C07302=1188.914,-2.420,-44.278,-179.914,5.732,148.990
C07303=1188.918,-2.670,-44.265,-179.916,5.731,148.990
C07304=1188.924,-2.919,-44.252,-179.918,5.732,148.991
C07305=1188.929,-3.170,-44.238,-179.921,5.731,148.992
C07306=1188.934,-3.418,-44.225,-179.923,5.731,148.992
C07307=1188.939,-3.668,-44.210,-179.926,5.730,148.993
C07308=1188.945,-3.918,-44.197,-179.928,5.729,148.993
C07309=1188.949,-4.167,-44.184,-179.931,5.729,148.994
C07310=1188.954,-4.417,-44.170,-179.934,5.728,148.995
C07311=1188.960,-4.666,-44.156,-179.936,5.727,148.995
C07312=1188.964,-4.916,-44.143,-179.938,5.727,148.996
C07313=1188.970,-5.165,-44.129,-179.941,5.726,148.997
C07314=1188.974,-5.415,-44.116,-179.944,5.726,148.997
C07315=1188.980,-5.664,-44.102,-179.946,5.725,148.998
C07316=1188.985,-5.915,-44.089,-179.948,5.725,148.999
C07317=1188.990,-6.163,-44.075,-179.951,5.725,148.999
C07318=1188.995,-6.414,-44.062,-179.953,5.725,149.000
C07319=1189.000,-6.663,-44.048,-179.955,5.724,149.000
C07320=1189.005,-6.913,-44.035,-179.958,5.723,149.001
C07321=1189.010,-7.162,-44.021,-179.961,5.723,149.002
C07322=1189.015,-7.412,-44.008,-179.963,5.722,149.002
C07323=1189.020,-7.661,-43.994,-179.966,5.721,149.003
C07324=1189.026,-7.911,-43.981,-179.968,5.721,149.004
C07325=1189.030,-8.161,-43.967,-179.971,5.720,149.004
C07326=1189.036,-8.410,-43.954,-179.974,5.720,149.005
C07327=1189.041,-8.660,-43.941,-179.975,5.720,149.005
C07328=1189.046,-8.909,-43.927,-179.978,5.719,149.006
C07329=1189.051,-9.159,-43.914,-179.980,5.719,149.007
C07330=1189.056,-9.408,-43.900,-179.983,5.719,149.008
C07331=1189.061,-9.658,-43.887,-179.986,5.718,149.008
C07332=1189.067,-9.908,-43.874,-179.988,5.717,149.009
C07333=1189.071,-10.157,-43.860,-179.991,5.717,149.009
C07334=1189.077,-10.407,-43.847,-179.993,5.716,149.010
C07335=1189.081,-10.657,-43.834,-179.996,5.716,149.011
C07336=1189.087,-10.906,-43.820,-179.997,5.716,149.011
C07337=1189.092,-11.156,-43.807,180.000,5.715,149.012
C07338=1189.097,-11.406,-43.794,179.997,5.715,149.013
C07339=1189.102,-11.654,-43.781,179.995,5.714,149.013
C07340=1189.108,-11.905,-43.767,179.992,5.714,149.014
C07341=1189.113,-12.154,-43.754,179.990,5.713,149.014
C07342=1189.118,-12.404,-43.740,179.987,5.713,149.015
C07343=1189.123,-12.653,-43.728,179.984,5.712,149.016
C07344=1189.127,-12.903,-43.715,179.983,5.712,149.016
C07345=1189.133,-13.153,-43.701,179.980,5.712,149.017
C07346=1189.137,-13.402,-43.688,179.978,5.711,149.018
C07347=1189.143,-13.652,-43.675,179.975,5.711,149.018
C07348=1189.148,-13.901,-43.662,179.973,5.710,149.019
C07349=1189.154,-14.151,-43.648,179.970,5.709,149.020
C07350=1189.158,-14.400,-43.635,179.967,5.709,149.020
C07351=1189.164,-14.650,-43.622,179.965,5.708,149.021
C07352=1189.169,-14.900,-43.609,179.963,5.708,149.021
C07353=1189.173,-15.150,-43.596,179.960,5.708,149.022
C07354=1189.179,-15.399,-43.583,179.958,5.707,149.023
C07355=1189.184,-15.648,-43.569,179.955,5.707,149.023
C07356=1189.189,-15.898,-43.556,179.953,5.707,149.024
C07357=1189.194,-16.148,-43.543,179.950,5.706,149.025
C07358=1189.199,-16.397,-43.531,179.948,5.705,149.025
C07359=1189.205,-16.647,-43.517,179.946,5.706,149.026
C07360=1189.210,-16.897,-43.504,179.943,5.705,149.027
C07361=1189.214,-17.146,-43.491,179.941,5.704,149.027
C07362=1189.220,-17.396,-43.478,179.938,5.704,149.028
C07363=1189.225,-17.645,-43.465,179.935,5.703,149.029
C07364=1189.230,-17.895,-43.452,179.933,5.703,149.029
C07365=1189.235,-18.145,-43.439,179.931,5.702,149.030
C07366=1189.241,-18.394,-43.426,179.929,5.702,149.030
C07367=1189.245,-18.644,-43.413,179.926,5.702,149.031
C07368=1189.251,-18.894,-43.400,179.923,5.701,149.032
C07369=1189.256,-19.143,-43.387,179.921,5.701,149.032
C07370=1189.260,-19.392,-43.374,179.918,5.700,149.033
C07371=1189.266,-19.642,-43.361,179.916,5.700,149.034
C07372=1189.271,-19.891,-43.348,179.914,5.700,149.034
C07373=1189.276,-20.141,-43.335,179.912,5.699,149.035
C07374=1189.282,-20.391,-43.322,179.909,5.699,149.036
C07375=1189.287,-20.640,-43.309,179.906,5.698,149.036
C07376=1189.291,-20.890,-43.296,179.904,5.698,149.037
C07377=1189.296,-21.139,-43.284,179.901,5.697,149.037
C07378=1189.302,-21.389,-43.270,179.899,5.696,149.038
C07379=1189.307,-21.639,-43.258,179.897,5.697,149.039
C07380=1189.312,-21.888,-43.245,179.894,5.696,149.039
C07381=1189.318,-22.138,-43.232,179.891,5.696,149.040
C07382=1189.322,-22.388,-43.219,179.889,5.695,149.041
C07383=1189.327,-22.637,-43.206,179.886,5.695,149.041
C07384=1189.333,-22.887,-43.194,179.884,5.694,149.042
C07385=1189.338,-23.157,-43.179,179.882,5.694,149.043
C07386=1189.343,-23.426,-43.166,179.879,5.694,149.043
C07387=1189.350,-23.696,-43.152,179.876,5.694,149.044
C07388=1189.355,-23.966,-43.138,179.874,5.693,149.045
C07389=1189.360,-24.215,-43.126,179.871,5.693,149.046
C07390=1189.365,-24.465,-43.114,179.869,5.692,149.046
C07391=1189.370,-24.715,-43.100,179.866,5.691,149.047
C07392=1189.376,-24.964,-43.087,179.864,5.691,149.047
C07393=1189.381,-25.214,-43.075,179.861,5.690,149.048
C07394=1189.386,-25.463,-43.062,179.859,5.690,149.049
C07395=1189.390,-25.713,-43.049,179.857,5.690,149.049
C07396=1189.396,-25.963,-43.036,179.854,5.689,149.050
C07397=1189.401,-26.212,-43.023,179.851,5.689,149.051
C07398=1189.407,-26.462,-43.012,179.849,5.688,149.051
C07399=1189.411,-26.712,-42.999,179.847,5.689,149.052
C07400=1189.416,-26.961,-42.986,179.844,5.688,149.052
C07401=1189.422,-27.211,-42.973,179.842,5.688,149.053
C07402=1189.427,-27.460,-42.961,179.840,5.687,149.054
C07403=1189.431,-27.710,-42.948,179.837,5.686,149.054
C07404=1189.437,-27.960,-42.935,179.835,5.687,149.055
C07405=1189.442,-28.210,-42.923,179.832,5.686,149.056
C07406=1189.448,-28.459,-42.910,179.830,5.685,149.056
C07407=1189.453,-28.708,-42.897,179.827,5.685,149.057
C07408=1189.457,-28.958,-42.885,179.825,5.684,149.058
C07409=1189.463,-29.208,-42.873,179.823,5.685,149.058
C07410=1189.468,-29.457,-42.860,179.820,5.684,149.059
C07411=1189.473,-29.707,-42.847,179.818,5.684,149.059
C07412=1189.478,-29.956,-42.835,179.815,5.683,149.060
C07413=1189.483,-30.207,-42.823,179.812,5.683,149.061
C07414=1189.489,-30.456,-42.809,179.810,5.683,149.062
C07415=1189.494,-30.706,-42.797,179.808,5.682,149.062
C07416=1189.499,-30.956,-42.785,179.806,5.682,149.063
C07417=1189.504,-31.205,-42.772,179.803,5.681,149.063
C07418=1189.509,-31.455,-42.759,179.800,5.681,149.064
C07419=1189.514,-31.704,-42.747,179.799,5.681,149.065
C07420=1189.519,-31.954,-42.735,179.796,5.680,149.065
C07421=1189.525,-32.204,-42.722,179.793,5.680,149.066
C07422=1189.530,-32.453,-42.710,179.791,5.679,149.067
C07423=1189.535,-32.703,-42.698,179.788,5.679,149.067
C07424=1189.540,-32.952,-42.685,179.786,5.679,149.068
C07425=1189.545,-33.202,-42.672,179.784,5.678,149.069
C07426=1189.550,-33.452,-42.660,179.781,5.678,149.069
C07427=1189.555,-33.701,-42.648,179.779,5.677,149.070
C07428=1189.561,-33.951,-42.636,179.776,5.677,149.070
C07429=1189.566,-34.201,-42.623,179.774,5.677,149.071
C07430=1189.571,-34.450,-42.611,179.772,5.677,149.072
C07431=1189.576,-34.700,-42.599,179.769,5.676,149.073
C07432=1189.582,-34.949,-42.586,179.767,5.675,149.073
C07433=1189.586,-35.200,-42.574,179.765,5.676,149.074
C07434=1189.592,-35.449,-42.561,179.762,5.675,149.074
C07435=1189.597,-35.698,-42.549,179.759,5.675,149.075
C07436=1189.602,-35.948,-42.537,179.757,5.674,149.076
C07437=1189.607,-36.198,-42.524,179.755,5.674,149.076
C07438=1189.613,-36.448,-42.512,179.752,5.674,149.077
C07439=1189.617,-36.697,-42.500,179.750,5.673,149.078
C07440=1189.622,-36.947,-42.488,179.748,5.673,149.078
C07441=1189.628,-37.196,-42.476,179.745,5.672,149.079
C07442=1189.633,-37.446,-42.464,179.743,5.672,149.080
C07443=1189.638,-37.695,-42.451,179.740,5.672,149.080
C07444=1189.644,-37.945,-42.439,179.738,5.671,149.081
C07445=1189.648,-38.195,-42.426,179.735,5.671,149.081
C07446=1189.654,-38.445,-42.415,179.733,5.671,149.082
C07447=1189.659,-38.694,-42.402,179.731,5.671,149.083
C07448=1189.664,-38.944,-42.390,179.728,5.670,149.083
C07449=1189.669,-39.194,-42.378,179.726,5.669,149.084
C07450=1189.674,-39.443,-42.366,179.724,5.670,149.085
C07451=1189.679,-39.693,-42.354,179.721,5.669,149.085
C07452=1189.684,-39.943,-42.342,179.719,5.668,149.086
C07453=1189.690,-40.192,-42.330,179.716,5.668,149.087
C07454=1189.695,-40.442,-42.317,179.714,5.668,149.087
C07455=1189.700,-40.692,-42.305,179.711,5.668,149.088
C07456=1189.706,-40.941,-42.293,179.709,5.667,149.088
C07457=1189.710,-41.191,-42.281,179.707,5.667,149.089
C07458=1189.716,-41.441,-42.270,179.704,5.667,149.090
C07459=1189.721,-41.690,-42.257,179.702,5.667,149.091
C07460=1189.726,-41.940,-42.245,179.700,5.666,149.091
C07461=1189.731,-42.189,-42.233,179.697,5.665,149.092
C07462=1189.736,-42.439,-42.221,179.695,5.666,149.092
C07463=1189.741,-42.689,-42.209,179.692,5.665,149.093
C07464=1189.747,-42.938,-42.197,179.690,5.665,149.094
C07465=1189.752,-43.188,-42.185,179.687,5.664,149.094
C07466=1189.757,-43.438,-42.173,179.685,5.664,149.095
C07467=1189.762,-43.687,-42.161,179.683,5.664,149.096
C07468=1189.767,-43.937,-42.149,179.680,5.663,149.096
C07469=1189.773,-44.187,-42.137,179.678,5.663,149.097
C07470=1189.778,-44.436,-42.125,179.676,5.663,149.098
C07471=1189.783,-44.686,-42.113,179.673,5.663,149.098
C07472=1189.788,-44.936,-42.101,179.670,5.662,149.099
C07473=1189.793,-45.186,-42.090,179.668,5.661,149.099
C07474=1189.799,-45.435,-42.077,179.666,5.662,149.100
C07475=1189.803,-45.685,-42.066,179.663,5.661,149.101
C07476=1189.809,-45.934,-42.054,179.661,5.661,149.102
C07477=1189.814,-46.184,-42.041,179.659,5.661,149.102
C07478=1189.819,-46.434,-42.029,179.657,5.660,149.103
C07479=1189.824,-46.683,-42.018,179.654,5.660,149.103
C07480=1189.829,-46.933,-42.006,179.651,5.659,149.104
C07481=1189.835,-47.183,-41.994,179.650,5.659,149.105
C07482=1189.839,-47.432,-41.982,179.647,5.659,149.105
C07483=1189.845,-47.681,-41.971,179.644,5.658,149.106
C07484=1189.851,-47.931,-41.959,179.642,5.658,149.107
C07485=1189.856,-48.181,-41.947,179.640,5.658,149.107
C07486=1189.861,-48.431,-41.936,179.637,5.658,149.108
C07487=1189.866,-48.680,-41.923,179.635,5.657,149.109
C07488=1189.871,-48.930,-41.911,179.633,5.657,149.109
C07489=1189.877,-49.201,-41.898,179.630,5.657,149.110
C07490=1189.883,-49.471,-41.886,179.628,5.656,149.110
C07491=1189.888,-49.741,-41.873,179.625,5.656,149.111
C07492=1189.893,-50.012,-41.860,179.622,5.655,149.112
C07493=1189.899,-50.260,-41.849,179.620,5.655,149.113
C07494=1189.904,-50.510,-41.838,179.618,5.655,149.113
C07495=1189.910,-50.760,-41.826,179.615,5.655,149.114
C07496=1189.914,-51.009,-41.814,179.613,5.654,149.114
C07497=1189.919,-51.259,-41.802,179.611,5.654,149.115
C07498=1189.925,-51.509,-41.790,179.608,5.654,149.116
C07499=1189.929,-51.759,-41.779,179.605,5.654,149.117
C07500=1189.935,-52.009,-41.767,179.603,5.653,149.117
C07501=1189.940,-52.258,-41.756,179.601,5.653,149.118
C07502=1189.946,-52.508,-41.744,179.598,5.653,149.118
C07503=1189.950,-52.757,-41.733,179.596,5.652,149.119
C07504=1189.956,-53.007,-41.721,179.594,5.652,149.120
C07505=1189.961,-53.257,-41.709,179.592,5.652,149.120
C07506=1189.966,-53.507,-41.698,179.589,5.651,149.121
C07507=1189.971,-53.757,-41.686,179.587,5.652,149.122
C07508=1189.977,-54.006,-41.675,179.585,5.651,149.122
C07509=1189.982,-54.256,-41.663,179.582,5.650,149.123
C07510=1189.987,-54.505,-41.652,179.579,5.650,149.124
C07511=1189.992,-54.755,-41.640,179.577,5.650,149.124
C07512=1189.997,-55.005,-41.628,179.575,5.650,149.125
C07513=1190.002,-55.255,-41.616,179.572,5.649,149.125
C07514=1190.008,-55.505,-41.605,179.570,5.649,149.126
C07515=1190.013,-55.754,-41.594,179.568,5.649,149.127
C07516=1190.018,-56.004,-41.582,179.565,5.648,149.127
C07517=1190.023,-56.253,-41.571,179.563,5.649,149.128
C07518=1190.029,-56.503,-41.559,179.561,5.648,149.129
C07519=1190.033,-56.753,-41.547,179.558,5.647,149.129
C07520=1190.039,-57.002,-41.536,179.556,5.648,149.130
C07521=1190.044,-57.252,-41.525,179.554,5.647,149.131
C07522=1190.049,-57.501,-41.513,179.551,5.647,149.131
C07523=1190.054,-57.751,-41.501,179.549,5.646,149.132
C07524=1190.059,-58.001,-41.490,179.547,5.646,149.133
C07525=1190.065,-58.250,-41.479,179.544,5.646,149.133
C07526=1190.070,-58.500,-41.468,179.541,5.645,149.134
C07527=1190.075,-58.750,-41.456,179.540,5.645,149.134
C07528=1190.080,-59.000,-41.445,179.537,5.645,149.135
C07529=1190.085,-59.250,-41.433,179.535,5.645,149.136
C07530=1190.091,-59.499,-41.422,179.532,5.645,149.137
C07531=1190.096,-59.749,-41.410,179.530,5.644,149.137
C07532=1190.101,-59.998,-41.399,179.528,5.644,149.138
C07533=1190.105,-60.248,-41.388,179.526,5.644,149.138
C07534=1190.112,-60.498,-41.377,179.523,5.643,149.139
C07535=1190.116,-60.747,-41.365,179.521,5.643,149.140
C07536=1190.122,-60.997,-41.354,179.519,5.643,149.140
C07537=1190.127,-61.247,-41.342,179.516,5.643,149.141
C07538=1190.132,-61.496,-41.331,179.514,5.642,149.142
C07539=1190.138,-61.746,-41.320,179.512,5.642,149.142
C07540=1190.142,-61.996,-41.309,179.509,5.642,149.143
C07541=1190.148,-62.246,-41.297,179.506,5.641,149.144
C07542=1190.153,-62.495,-41.286,179.505,5.641,149.144
C07543=1190.158,-62.744,-41.275,179.502,5.641,149.145
C07544=1190.163,-62.995,-41.264,179.499,5.641,149.146
C07545=1190.169,-63.244,-41.253,179.498,5.641,149.146
C07546=1190.174,-63.494,-41.241,179.495,5.640,149.147
C07547=1190.179,-63.744,-41.229,179.492,5.640,149.147
C07548=1190.184,-63.994,-41.219,179.490,5.640,149.148
C07549=1190.190,-64.243,-41.207,179.488,5.639,149.149
C07550=1190.195,-64.493,-41.196,179.486,5.639,149.149
C07551=1190.200,-64.743,-41.186,179.483,5.639,149.150
C07552=1190.206,-64.992,-41.174,179.481,5.639,149.151
C07553=1190.210,-65.242,-41.163,179.479,5.638,149.151
C07554=1190.215,-65.492,-41.152,179.477,5.638,149.152
C07555=1190.221,-65.741,-41.141,179.474,5.638,149.153
C07556=1190.226,-65.991,-41.129,179.472,5.637,149.153
C07557=1190.231,-66.241,-41.119,179.470,5.638,149.154
C07558=1190.236,-66.490,-41.108,179.467,5.637,149.154
C07559=1190.242,-66.740,-41.096,179.464,5.637,149.155
C07560=1190.247,-66.990,-41.085,179.463,5.637,149.156
C07561=1190.252,-67.239,-41.074,179.460,5.636,149.156
C07562=1190.257,-67.489,-41.063,179.457,5.636,149.157
C07563=1190.262,-67.739,-41.052,179.456,5.636,149.158
C07564=1190.268,-67.988,-41.041,179.453,5.635,149.158
C07565=1190.272,-68.238,-41.030,179.451,5.636,149.159
C07566=1190.278,-68.488,-41.019,179.448,5.635,149.160
C07567=1190.284,-68.737,-41.008,179.446,5.635,149.160
C07568=1190.289,-68.988,-40.997,179.444,5.635,149.161
C07569=1190.295,-69.237,-40.986,179.441,5.634,149.162
C07570=1190.299,-69.486,-40.974,179.439,5.634,149.162
C07571=1190.304,-69.737,-40.964,179.437,5.634,149.163
C07572=1190.310,-69.986,-40.953,179.434,5.634,149.163
C07573=1190.315,-70.236,-40.942,179.432,5.633,149.164
C07574=1190.320,-70.486,-40.930,179.430,5.633,149.165
C07575=1190.326,-70.735,-40.920,179.427,5.633,149.165
C07576=1190.330,-70.985,-40.909,179.425,5.633,149.166
C07577=1190.336,-71.234,-40.899,179.423,5.632,149.167
C07578=1190.341,-71.484,-40.887,179.421,5.632,149.167
C07579=1190.346,-71.735,-40.876,179.418,5.632,149.168
C07580=1190.352,-71.984,-40.865,179.416,5.632,149.169
C07581=1190.357,-72.234,-40.855,179.414,5.631,149.169
C07582=1190.362,-72.483,-40.844,179.412,5.631,149.170
C07583=1190.368,-72.733,-40.833,179.409,5.631,149.171
C07584=1190.373,-72.982,-40.822,179.407,5.630,149.171
C07585=1190.378,-73.232,-40.811,179.405,5.631,149.172
C07586=1190.383,-73.482,-40.800,179.402,5.630,149.172
C07587=1190.388,-73.732,-40.790,179.400,5.631,149.173
C07588=1190.393,-73.981,-40.778,179.398,5.630,149.174
C07589=1190.398,-74.231,-40.768,179.395,5.629,149.174
C07590=1190.404,-74.481,-40.757,179.393,5.630,149.175
C07591=1190.409,-74.730,-40.746,179.391,5.629,149.176
C07592=1190.414,-74.981,-40.735,179.388,5.628,149.176
C07593=1190.420,-75.252,-40.723,179.386,5.629,149.177
C07594=1190.426,-75.521,-40.712,179.383,5.628,149.178
C07595=1190.431,-75.793,-40.700,179.381,5.628,149.178
C07596=1190.437,-76.064,-40.688,179.378,5.628,149.179
C07597=1190.443,-76.314,-40.678,179.376,5.628,149.180
C07598=1190.447,-76.563,-40.667,179.374,5.627,149.180
C07599=1190.453,-76.813,-40.656,179.372,5.628,149.181
C07600=1190.458,-77.063,-40.646,179.369,5.627,149.182
C07601=1190.463,-77.312,-40.635,179.367,5.626,149.182
C07602=1190.468,-77.562,-40.624,179.365,5.627,149.183
C07603=1190.474,-77.812,-40.614,179.362,5.626,149.184
C07604=1190.479,-78.061,-40.603,179.360,5.626,149.184
C07605=1190.484,-78.311,-40.593,179.358,5.626,149.185
C07606=1190.490,-78.561,-40.581,179.355,5.625,149.186
C07607=1190.495,-78.810,-40.571,179.353,5.625,149.186
C07608=1190.500,-79.061,-40.560,179.351,5.625,149.187
C07609=1190.506,-79.310,-40.550,179.348,5.625,149.187
C07610=1190.510,-79.560,-40.538,179.347,5.625,149.188
C07611=1190.516,-79.809,-40.528,179.344,5.624,149.189
C07612=1190.521,-80.060,-40.518,179.342,5.625,149.189
C07613=1190.527,-80.309,-40.507,179.339,5.624,149.190
C07614=1190.531,-80.559,-40.496,179.337,5.623,149.190
C07615=1190.537,-80.808,-40.486,179.335,5.624,149.191
C07616=1190.542,-81.059,-40.475,179.332,5.623,149.192
C07617=1190.548,-81.308,-40.465,179.331,5.623,149.192
C07618=1190.553,-81.557,-40.454,179.328,5.623,149.193
C07619=1190.558,-81.807,-40.444,179.325,5.622,149.194
C07620=1190.563,-82.057,-40.433,179.324,5.622,149.194
C07621=1190.568,-82.307,-40.423,179.321,5.622,149.195
C07622=1190.574,-82.557,-40.413,179.319,5.622,149.196
C07623=1190.579,-82.806,-40.401,179.317,5.622,149.196
C07624=1190.584,-83.056,-40.391,179.315,5.622,149.197
C07625=1190.589,-83.306,-40.381,179.312,5.622,149.198
C07626=1190.595,-83.556,-40.370,179.310,5.621,149.198
C07627=1190.601,-83.805,-40.360,179.308,5.621,149.199
C07628=1190.604,-84.054,-40.349,179.305,5.621,149.200
C07629=1190.610,-84.304,-40.339,179.303,5.621,149.200
C07630=1190.615,-84.554,-40.329,179.301,5.620,149.201
C07631=1190.621,-84.804,-40.319,179.298,5.620,149.201
C07632=1190.626,-85.054,-40.308,179.296,5.620,149.202
C07633=1190.631,-85.304,-40.298,179.294,5.620,149.203
C07634=1190.637,-85.553,-40.288,179.292,5.620,149.203
C07635=1190.642,-85.803,-40.276,179.289,5.619,149.204
C07636=1190.647,-86.052,-40.266,179.287,5.619,149.205
C07637=1190.652,-86.302,-40.255,179.285,5.619,149.205
C07638=1190.658,-86.552,-40.245,179.283,5.618,149.206
C07639=1190.663,-86.801,-40.236,179.280,5.619,149.206
C07640=1190.668,-87.052,-40.225,179.278,5.618,149.207
C07641=1190.673,-87.301,-40.215,179.276,5.618,149.208
C07642=1190.678,-87.551,-40.204,179.274,5.618,149.208
C07643=1190.684,-87.801,-40.194,179.271,5.617,149.209
C07644=1190.689,-88.050,-40.184,179.269,5.617,149.209
C07645=1190.694,-88.301,-40.173,179.267,5.617,149.210
C07646=1190.700,-88.550,-40.163,179.264,5.617,149.211
C07647=1190.705,-88.799,-40.153,179.262,5.617,149.211
C07648=1190.710,-89.050,-40.143,179.260,5.616,149.212
C07649=1190.715,-89.299,-40.133,179.258,5.617,149.213
C07650=1190.720,-89.549,-40.122,179.255,5.616,149.213
C07651=1190.726,-89.798,-40.111,179.253,5.616,149.214
C07652=1190.731,-90.048,-40.101,179.251,5.616,149.215
C07653=1190.736,-90.298,-40.092,179.249,5.616,149.215
C07654=1190.742,-90.548,-40.081,179.246,5.615,149.216
C07655=1190.747,-90.798,-40.071,179.244,5.615,149.217
C07656=1190.752,-91.048,-40.061,179.242,5.615,149.217
C07657=1190.758,-91.297,-40.050,179.239,5.615,149.218
C07658=1190.763,-91.547,-40.041,179.237,5.615,149.219
C07659=1190.768,-91.797,-40.030,179.235,5.614,149.219
C07660=1190.773,-92.046,-40.020,179.233,5.615,149.220
C07661=1190.779,-92.296,-40.010,179.230,5.614,149.220
C07662=1190.784,-92.546,-39.999,179.229,5.614,149.221
C07663=1190.789,-92.795,-39.990,179.226,5.614,149.222
C07664=1190.794,-93.045,-39.979,179.223,5.613,149.222
C07665=1190.799,-93.295,-39.969,179.222,5.613,149.223
C07666=1190.805,-93.545,-39.959,179.219,5.613,149.224
C07667=1190.810,-93.794,-39.949,179.217,5.613,149.224
C07668=1190.815,-94.043,-39.939,179.215,5.613,149.225
C07669=1190.821,-94.294,-39.929,179.213,5.613,149.225
C07670=1190.826,-94.544,-39.919,179.210,5.613,149.226
C07671=1190.831,-94.793,-39.909,179.209,5.613,149.227
C07672=1190.836,-95.043,-39.899,179.206,5.612,149.227
C07673=1190.842,-95.293,-39.888,179.204,5.611,149.228
C07674=1190.847,-95.542,-39.878,179.202,5.612,149.229
C07675=1190.852,-95.792,-39.869,179.199,5.611,149.229
C07676=1190.857,-96.043,-39.859,179.197,5.611,149.230
C07677=1190.863,-96.292,-39.849,179.195,5.611,149.230
C07678=1190.868,-96.541,-39.839,179.193,5.611,149.231
C07679=1190.873,-96.791,-39.829,179.190,5.611,149.232
C07680=1190.878,-97.041,-39.818,179.188,5.611,149.232
C07681=1190.884,-97.291,-39.808,179.186,5.611,149.233
C07682=1190.889,-97.540,-39.799,179.183,5.610,149.234
C07683=1190.895,-97.790,-39.789,179.181,5.610,149.234
C07684=1190.900,-98.040,-39.778,179.179,5.609,149.235
C07685=1190.905,-98.290,-39.769,179.177,5.610,149.235
C07686=1190.911,-98.540,-39.759,179.174,5.609,149.236
C07687=1190.916,-98.789,-39.749,179.173,5.609,149.237
C07688=1190.920,-99.039,-39.739,179.170,5.609,149.237
C07689=1190.926,-99.289,-39.729,179.168,5.609,149.238
C07690=1190.932,-99.539,-39.719,179.166,5.609,149.239
C07691=1190.937,-99.788,-39.710,179.164,5.609,149.239
C07692=1190.942,-100.038,-39.699,179.162,5.608,149.240
C07693=1190.947,-100.288,-39.689,179.159,5.608,149.240
C07694=1190.953,-100.538,-39.680,179.157,5.608,149.241
C07695=1190.958,-100.787,-39.670,179.155,5.607,149.242
C07696=1190.963,-101.037,-39.660,179.153,5.608,149.242
C07697=1190.969,-101.309,-39.649,179.150,5.607,149.243
C07698=1190.974,-101.580,-39.638,179.148,5.608,149.244
C07699=1190.980,-101.852,-39.628,179.146,5.607,149.244
C07700=1190.986,-102.123,-39.617,179.143,5.607,149.245
C07701=1190.991,-102.373,-39.608,179.141,5.607,149.246
C07702=1190.997,-102.623,-39.597,179.138,5.607,149.246
C07703=1191.001,-102.872,-39.588,179.137,5.607,149.247
C07704=1191.007,-103.122,-39.578,179.134,5.606,149.248
C07705=1191.012,-103.372,-39.569,179.132,5.606,149.248
C07706=1191.018,-103.621,-39.559,179.130,5.606,149.249
C07707=1191.022,-103.872,-39.549,179.127,5.605,149.250
C07708=1191.028,-104.121,-39.539,179.125,5.605,149.250
C07709=1191.034,-104.371,-39.530,179.123,5.605,149.251
C07710=1191.039,-104.621,-39.520,179.121,5.605,149.251
C07711=1191.044,-104.870,-39.510,179.118,5.605,149.252
C07712=1191.050,-105.120,-39.501,179.116,5.605,149.253
C07713=1191.055,-105.370,-39.490,179.114,5.604,149.253
C07714=1191.060,-105.620,-39.481,179.112,5.605,149.254
C07715=1191.065,-105.870,-39.471,179.110,5.604,149.254
C07716=1191.070,-106.119,-39.462,179.108,5.604,149.255
C07717=1191.076,-106.369,-39.452,179.105,5.604,149.256
C07718=1191.081,-106.618,-39.442,179.103,5.604,149.256
C07719=1191.087,-106.868,-39.433,179.101,5.603,149.257
C07720=1191.091,-107.118,-39.423,179.099,5.603,149.257
C07721=1191.097,-107.369,-39.414,179.096,5.603,149.258
C07722=1191.102,-107.618,-39.404,179.094,5.603,149.259
C07723=1191.108,-107.868,-39.394,179.092,5.603,149.259
C07724=1191.113,-108.117,-39.385,179.090,5.603,149.260
C07725=1191.119,-108.367,-39.375,179.088,5.602,149.261
C07726=1191.123,-108.617,-39.366,179.086,5.603,149.261
C07727=1191.129,-108.867,-39.356,179.083,5.602,149.262
C07728=1191.134,-109.116,-39.347,179.081,5.601,149.262
C07729=1191.139,-109.366,-39.338,179.079,5.602,149.263
C07730=1191.144,-109.616,-39.327,179.077,5.601,149.264
C07731=1191.149,-109.866,-39.318,179.075,5.601,149.264
C07732=1191.155,-110.115,-39.308,179.072,5.601,149.265
C07733=1191.160,-110.365,-39.299,179.070,5.601,149.266
C07734=1191.166,-110.615,-39.289,179.068,5.601,149.266
C07735=1191.171,-110.865,-39.280,179.066,5.601,149.267
C07736=1191.177,-111.114,-39.270,179.063,5.600,149.268
C07737=1191.182,-111.364,-39.261,179.062,5.600,149.268
C07738=1191.187,-111.614,-39.252,179.059,5.600,149.269
C07739=1191.193,-111.863,-39.242,179.057,5.600,149.269
C07740=1191.198,-112.113,-39.233,179.055,5.600,149.270
C07741=1191.203,-112.363,-39.223,179.053,5.600,149.271
C07742=1191.208,-112.613,-39.214,179.051,5.599,149.271
C07743=1191.214,-112.863,-39.205,179.048,5.600,149.272
C07744=1191.219,-113.113,-39.194,179.046,5.599,149.273
C07745=1191.224,-113.363,-39.185,179.044,5.599,149.273
C07746=1191.229,-113.612,-39.176,179.041,5.599,149.274
C07747=1191.235,-113.862,-39.166,179.040,5.599,149.274
C07748=1191.240,-114.112,-39.157,179.037,5.598,149.275
C07749=1191.245,-114.361,-39.147,179.036,5.598,149.275
C07750=1191.250,-114.611,-39.138,179.033,5.598,149.276
C07751=1191.256,-114.861,-39.129,179.031,5.598,149.277
C07752=1191.261,-115.111,-39.119,179.029,5.598,149.277
C07753=1191.266,-115.361,-39.110,179.027,5.598,149.278
C07754=1191.272,-115.610,-39.101,179.024,5.597,149.279
C07755=1191.277,-115.860,-39.091,179.022,5.598,149.279
C07756=1191.282,-116.110,-39.082,179.020,5.597,149.280
C07757=1191.288,-116.360,-39.073,179.018,5.597,149.280
C07758=1191.293,-116.610,-39.064,179.016,5.597,149.281
C07759=1191.298,-116.859,-39.054,179.014,5.597,149.282
C07760=1191.303,-117.109,-39.045,179.011,5.597,149.282
C07761=1191.309,-117.359,-39.036,179.009,5.597,149.283
C07762=1191.314,-117.608,-39.026,179.007,5.596,149.284
C07763=1191.319,-117.858,-39.017,179.005,5.596,149.284
C07764=1191.325,-118.108,-39.008,179.003,5.596,149.285
C07765=1191.330,-118.358,-38.999,179.001,5.596,149.285
C07766=1191.335,-118.607,-38.989,178.998,5.595,149.286
C07767=1191.340,-118.857,-38.980,178.997,5.595,149.286
C07768=1191.346,-119.107,-38.971,178.994,5.595,149.287
C07769=1191.352,-119.357,-38.962,178.992,5.595,149.288
C07770=1191.357,-119.607,-38.953,178.990,5.595,149.288
C07771=1191.362,-119.856,-38.944,178.988,5.595,149.289
C07772=1191.367,-120.107,-38.934,178.986,5.595,149.290
C07773=1191.373,-120.356,-38.926,178.983,5.595,149.290
C07774=1191.378,-120.606,-38.917,178.982,5.595,149.291
C07775=1191.384,-120.855,-38.908,178.979,5.594,149.292
C07776=1191.388,-121.105,-38.898,178.977,5.594,149.292
C07777=1191.394,-121.355,-38.889,178.975,5.594,149.293
C07778=1191.400,-121.605,-38.880,178.973,5.594,149.293
C07779=1191.405,-121.854,-38.871,178.970,5.594,149.294
C07780=1191.410,-122.104,-38.862,178.969,5.594,149.294
C07781=1191.416,-122.354,-38.852,178.966,5.593,149.295
C07782=1191.421,-122.604,-38.843,178.965,5.593,149.296
C07783=1191.426,-122.854,-38.834,178.962,5.593,149.296
C07784=1191.431,-123.103,-38.825,178.960,5.593,149.297
C07785=1191.436,-123.353,-38.816,178.958,5.592,149.298
C07786=1191.442,-123.603,-38.807,178.956,5.593,149.298
C07787=1191.447,-123.853,-38.798,178.953,5.592,149.299
C07788=1191.453,-124.102,-38.789,178.951,5.593,149.299
C07789=1191.458,-124.352,-38.780,178.949,5.592,149.300
C07790=1191.463,-124.602,-38.771,178.947,5.592,149.301
C07791=1191.468,-124.851,-38.762,178.945,5.591,149.301
C07792=1191.474,-125.102,-38.752,178.943,5.592,149.302
C07793=1191.479,-125.351,-38.743,178.941,5.591,149.302
C07794=1191.484,-125.601,-38.735,178.938,5.591,149.303
C07795=1191.490,-125.851,-38.726,178.937,5.591,149.304
C07796=1191.495,-126.101,-38.717,178.934,5.591,149.304
C07797=1191.500,-126.350,-38.708,178.933,5.591,149.305
C07798=1191.506,-126.600,-38.699,178.930,5.591,149.305
C07799=1191.512,-126.850,-38.690,178.928,5.591,149.306
C07800=1191.517,-127.100,-38.681,178.926,5.590,149.307
C07801=1191.095,-127.111,-38.720,178.922,5.594,149.309
C07802=1191.090,-126.861,-38.729,178.924,5.594,149.308
C07803=1191.084,-126.611,-38.738,178.926,5.594,149.307
C07804=1191.079,-126.361,-38.747,178.929,5.594,149.307
C07805=1191.074,-126.111,-38.756,178.930,5.594,149.306
C07806=1191.068,-125.862,-38.764,178.933,5.595,149.305
C07807=1191.063,-125.612,-38.773,178.935,5.595,149.305
C07808=1191.058,-125.363,-38.783,178.937,5.595,149.304
C07809=1191.052,-125.113,-38.792,178.939,5.595,149.304
C07810=1191.047,-124.863,-38.801,178.941,5.595,149.303
C07811=1191.042,-124.613,-38.810,178.943,5.595,149.302
C07812=1191.037,-124.363,-38.819,178.946,5.596,149.302
C07813=1191.032,-124.113,-38.828,178.947,5.596,149.301
C07814=1191.026,-123.863,-38.837,178.949,5.595,149.301
C07815=1191.021,-123.613,-38.846,178.952,5.596,149.300
C07816=1191.015,-123.364,-38.855,178.954,5.596,149.299
C07817=1191.010,-123.114,-38.864,178.956,5.596,149.299
C07818=1191.004,-122.865,-38.873,178.958,5.596,149.298
C07819=1191.000,-122.615,-38.882,178.960,5.597,149.298
C07820=1190.994,-122.365,-38.892,178.962,5.596,149.297
C07821=1190.989,-122.115,-38.901,178.964,5.597,149.296
C07822=1190.983,-121.865,-38.910,178.967,5.597,149.296
C07823=1190.978,-121.616,-38.919,178.969,5.598,149.295
C07824=1190.972,-121.365,-38.928,178.971,5.597,149.295
C07825=1190.967,-121.116,-38.937,178.973,5.598,149.294
C07826=1190.962,-120.866,-38.947,178.975,5.598,149.293
C07827=1190.957,-120.616,-38.955,178.978,5.598,149.293
C07828=1190.952,-120.367,-38.964,178.979,5.598,149.292
C07829=1190.946,-120.116,-38.974,178.982,5.598,149.291
C07830=1190.941,-119.867,-38.983,178.984,5.598,149.291
C07831=1190.935,-119.618,-38.992,178.986,5.599,149.290
C07832=1190.930,-119.368,-39.001,178.988,5.599,149.290
C07833=1190.924,-119.118,-39.010,178.991,5.599,149.289
C07834=1190.919,-118.868,-39.019,178.992,5.599,149.289
C07835=1190.914,-118.618,-39.028,178.995,5.599,149.288
C07836=1190.909,-118.369,-39.038,178.997,5.599,149.287
C07837=1190.903,-118.119,-39.047,178.999,5.600,149.287
C07838=1190.898,-117.869,-39.056,179.001,5.599,149.286
C07839=1190.893,-117.619,-39.065,179.003,5.600,149.285
C07840=1190.887,-117.370,-39.075,179.006,5.600,149.285
C07841=1190.882,-117.120,-39.084,179.008,5.601,149.284
C07842=1190.877,-116.870,-39.093,179.010,5.600,149.284
C07843=1190.872,-116.621,-39.103,179.012,5.601,149.283
C07844=1190.866,-116.371,-39.112,179.014,5.600,149.282
C07845=1190.861,-116.121,-39.121,179.016,5.601,149.282
C07846=1190.856,-115.871,-39.130,179.018,5.601,149.281
C07847=1190.850,-115.621,-39.140,179.021,5.602,149.281
C07848=1190.845,-115.372,-39.149,179.023,5.601,149.280
C07849=1190.840,-115.122,-39.158,179.025,5.601,149.279
C07850=1190.834,-114.872,-39.168,179.027,5.602,149.279
C07851=1190.829,-114.622,-39.177,179.029,5.601,149.278
C07852=1190.823,-114.372,-39.187,179.031,5.602,149.278
C07853=1190.818,-114.123,-39.196,179.033,5.602,149.277
C07854=1190.813,-113.873,-39.205,179.035,5.602,149.276
C07855=1190.807,-113.623,-39.215,179.038,5.602,149.276
C07856=1190.803,-113.374,-39.224,179.040,5.602,149.275
C07857=1190.797,-113.124,-39.233,179.042,5.603,149.274
C07858=1190.792,-112.873,-39.243,179.045,5.603,149.274
C07859=1190.787,-112.624,-39.253,179.047,5.604,149.273
C07860=1190.781,-112.374,-39.262,179.049,5.603,149.272
C07861=1190.776,-112.124,-39.272,179.051,5.604,149.272
C07862=1190.771,-111.874,-39.281,179.053,5.604,149.271
C07863=1190.765,-111.624,-39.290,179.056,5.604,149.271
C07864=1190.760,-111.375,-39.300,179.057,5.604,149.270
C07865=1190.755,-111.125,-39.309,179.060,5.604,149.269
C07866=1190.750,-110.876,-39.319,179.062,5.604,149.269
C07867=1190.745,-110.626,-39.328,179.064,5.605,149.268
C07868=1190.739,-110.376,-39.338,179.066,5.605,149.268
C07869=1190.734,-110.126,-39.347,179.069,5.605,149.267
C07870=1190.728,-109.877,-39.357,179.071,5.605,149.266
C07871=1190.723,-109.627,-39.366,179.073,5.605,149.266
C07872=1190.717,-109.377,-39.375,179.075,5.605,149.265
C07873=1190.713,-109.127,-39.385,179.077,5.606,149.265
C07874=1190.708,-108.877,-39.394,179.079,5.605,149.264
C07875=1190.702,-108.628,-39.404,179.082,5.606,149.263
C07876=1190.697,-108.378,-39.413,179.084,5.606,149.263
C07877=1190.691,-108.128,-39.424,179.086,5.606,149.262
C07878=1190.686,-107.878,-39.432,179.088,5.606,149.261
C07879=1190.681,-107.629,-39.443,179.090,5.607,149.261
C07880=1190.675,-107.379,-39.452,179.092,5.607,149.260
C07881=1190.670,-107.129,-39.462,179.095,5.607,149.260
C07882=1190.665,-106.879,-39.471,179.097,5.607,149.259
C07883=1190.660,-106.629,-39.481,179.099,5.607,149.258
C07884=1190.655,-106.380,-39.491,179.101,5.607,149.258
C07885=1190.649,-106.130,-39.500,179.103,5.608,149.257
C07886=1190.644,-105.881,-39.510,179.105,5.607,149.256
C07887=1190.638,-105.630,-39.519,179.108,5.608,149.256
C07888=1190.633,-105.381,-39.529,179.110,5.608,149.255
C07889=1190.627,-105.131,-39.539,179.112,5.608,149.255
C07890=1190.623,-104.881,-39.549,179.114,5.608,149.254
C07891=1190.617,-104.632,-39.559,179.117,5.609,149.253
C07892=1190.612,-104.382,-39.568,179.119,5.609,149.253
C07893=1190.607,-104.132,-39.578,179.121,5.609,149.252
C07894=1190.602,-103.882,-39.587,179.124,5.609,149.251
C07895=1190.596,-103.633,-39.597,179.125,5.609,149.251
C07896=1190.591,-103.383,-39.608,179.128,5.610,149.250
C07897=1190.586,-103.133,-39.616,179.130,5.609,149.250
C07898=1190.580,-102.883,-39.627,179.132,5.610,149.249
C07899=1190.575,-102.634,-39.636,179.134,5.610,149.248
C07900=1190.569,-102.384,-39.646,179.136,5.610,149.248
C07901=1190.565,-102.134,-39.656,179.138,5.610,149.247
C07902=1190.558,-101.862,-39.666,179.141,5.610,149.246
C07903=1190.553,-101.591,-39.677,179.144,5.611,149.246
C07904=1190.548,-101.319,-39.687,179.146,5.610,149.245
C07905=1190.542,-101.047,-39.699,179.148,5.611,149.244
C07906=1190.537,-100.798,-39.708,179.151,5.612,149.244
C07907=1190.531,-100.548,-39.718,179.153,5.611,149.243
C07908=1190.525,-100.299,-39.728,179.155,5.612,149.243
C07909=1190.521,-100.049,-39.738,179.157,5.612,149.242
C07910=1190.515,-99.798,-39.748,179.160,5.612,149.241
C07911=1190.510,-99.549,-39.757,179.161,5.612,149.241
C07912=1190.505,-99.300,-39.767,179.164,5.612,149.240
C07913=1190.499,-99.050,-39.778,179.166,5.612,149.239
C07914=1190.494,-98.800,-39.787,179.168,5.613,149.239
C07915=1190.489,-98.550,-39.797,179.170,5.612,149.238
C07916=1190.483,-98.300,-39.807,179.173,5.613,149.238
C07917=1190.479,-98.051,-39.817,179.175,5.614,149.237
C07918=1190.473,-97.801,-39.826,179.177,5.613,149.236
C07919=1190.468,-97.551,-39.837,179.180,5.614,149.236
C07920=1190.463,-97.302,-39.847,179.182,5.614,149.235
C07921=1190.457,-97.052,-39.857,179.184,5.614,149.234
C07922=1190.452,-96.803,-39.867,179.186,5.614,149.234
C07923=1190.447,-96.552,-39.876,179.189,5.614,149.233
C07924=1190.441,-96.302,-39.887,179.190,5.614,149.233
C07925=1190.436,-96.053,-39.897,179.193,5.615,149.232
C07926=1190.430,-95.803,-39.907,179.195,5.614,149.231
C07927=1190.426,-95.553,-39.917,179.197,5.615,149.231
C07928=1190.420,-95.304,-39.927,179.200,5.616,149.230
C07929=1190.414,-95.054,-39.937,179.202,5.615,149.229
C07930=1190.410,-94.804,-39.946,179.204,5.616,149.229
C07931=1190.405,-94.554,-39.957,179.206,5.616,149.228
C07932=1190.399,-94.305,-39.967,179.208,5.616,149.228
C07933=1190.393,-94.055,-39.977,179.210,5.616,149.227
C07934=1190.389,-93.805,-39.987,179.213,5.616,149.226
C07935=1190.384,-93.556,-39.997,179.215,5.617,149.226
C07936=1190.378,-93.306,-40.008,179.217,5.617,149.225
C07937=1190.373,-93.055,-40.018,179.220,5.617,149.224
C07938=1190.368,-92.806,-40.027,179.222,5.617,149.224
C07939=1190.362,-92.556,-40.037,179.224,5.618,149.223
C07940=1190.357,-92.307,-40.048,179.226,5.617,149.222
C07941=1190.352,-92.057,-40.058,179.229,5.618,149.222
C07942=1190.346,-91.807,-40.068,179.231,5.618,149.221
C07943=1190.341,-91.558,-40.078,179.233,5.618,149.220
C07944=1190.336,-91.308,-40.089,179.236,5.619,149.220
C07945=1190.331,-91.058,-40.099,179.238,5.619,149.219
C07946=1190.325,-90.809,-40.109,179.240,5.619,149.218
C07947=1190.320,-90.558,-40.120,179.242,5.619,149.218
C07948=1190.315,-90.309,-40.129,179.245,5.619,149.217
C07949=1190.309,-90.060,-40.139,179.246,5.619,149.217
C07950=1190.304,-89.809,-40.150,179.249,5.620,149.216
C07951=1190.299,-89.560,-40.160,179.252,5.620,149.215
C07952=1190.293,-89.310,-40.170,179.253,5.620,149.215
C07953=1190.289,-89.060,-40.180,179.256,5.621,149.214
C07954=1190.283,-88.811,-40.191,179.258,5.620,149.213
C07955=1190.278,-88.561,-40.201,179.260,5.621,149.213
C07956=1190.273,-88.311,-40.211,179.262,5.621,149.212
C07957=1190.267,-88.061,-40.222,179.265,5.621,149.212
C07958=1190.262,-87.811,-40.232,179.267,5.622,149.211
C07959=1190.257,-87.562,-40.242,179.269,5.621,149.210
C07960=1190.252,-87.312,-40.252,179.272,5.622,149.210
C07961=1190.247,-87.062,-40.262,179.273,5.622,149.209
C07962=1190.241,-86.813,-40.273,179.276,5.622,149.208
C07963=1190.236,-86.562,-40.283,179.278,5.622,149.208
C07964=1190.231,-86.313,-40.294,179.280,5.623,149.207
C07965=1190.225,-86.064,-40.304,179.283,5.623,149.207
C07966=1190.220,-85.814,-40.315,179.285,5.623,149.206
C07967=1190.215,-85.564,-40.325,179.287,5.623,149.205
C07968=1190.210,-85.314,-40.336,179.289,5.623,149.205
C07969=1190.204,-85.064,-40.346,179.292,5.623,149.204
C07970=1190.199,-84.815,-40.356,179.294,5.624,149.203
C07971=1190.194,-84.565,-40.366,179.296,5.624,149.203
C07972=1190.189,-84.315,-40.376,179.299,5.624,149.202
C07973=1190.184,-84.066,-40.388,179.301,5.624,149.202
C07974=1190.178,-83.816,-40.398,179.303,5.625,149.201
C07975=1190.173,-83.566,-40.408,179.306,5.625,149.200
C07976=1190.168,-83.316,-40.419,179.308,5.625,149.200
C07977=1190.162,-83.067,-40.429,179.310,5.626,149.199
C07978=1190.157,-82.817,-40.440,179.312,5.625,149.198
C07979=1190.152,-82.568,-40.450,179.314,5.626,149.198
C07980=1190.147,-82.317,-40.461,179.317,5.626,149.197
C07981=1190.141,-82.068,-40.471,179.319,5.626,149.196
C07982=1190.136,-81.818,-40.482,179.322,5.626,149.196
C07983=1190.131,-81.569,-40.493,179.323,5.626,149.195
C07984=1190.126,-81.318,-40.503,179.326,5.627,149.194
C07985=1190.120,-81.069,-40.513,179.329,5.627,149.194
C07986=1190.115,-80.819,-40.524,179.330,5.627,149.193
C07987=1190.110,-80.570,-40.535,179.333,5.628,149.193
C07988=1190.105,-80.319,-40.545,179.335,5.627,149.192
C07989=1190.099,-80.070,-40.556,179.337,5.628,149.191
C07990=1190.094,-79.820,-40.566,179.340,5.629,149.191
C07991=1190.089,-79.571,-40.577,179.342,5.628,149.190
C07992=1190.084,-79.321,-40.587,179.344,5.629,149.189
C07993=1190.079,-79.071,-40.598,179.346,5.629,149.189
C07994=1190.073,-78.821,-40.608,179.349,5.629,149.188
C07995=1190.068,-78.572,-40.619,179.351,5.630,149.188
C07996=1190.063,-78.322,-40.630,179.353,5.629,149.187
C07997=1190.058,-78.072,-40.640,179.356,5.630,149.186
C07998=1190.052,-77.823,-40.651,179.358,5.630,149.186
C07999=1190.047,-77.573,-40.662,179.360,5.630,149.185
C08000=1190.042,-77.323,-40.672,179.363,5.631,149.184
C08001=1190.037,-77.074,-40.683,179.365,5.630,149.184
C08002=1190.031,-76.824,-40.694,179.367,5.631,149.183
C08003=1190.026,-76.574,-40.705,179.369,5.631,149.182
C08004=1190.021,-76.325,-40.716,179.372,5.631,149.182
C08005=1190.016,-76.074,-40.726,179.374,5.632,149.181
C08006=1190.010,-75.803,-40.738,179.376,5.632,149.180
C08007=1190.004,-75.533,-40.749,179.379,5.632,149.180
C08008=1189.998,-75.262,-40.761,179.382,5.632,149.179
C08009=1189.993,-74.991,-40.773,179.384,5.633,149.178
C08010=1189.987,-74.741,-40.784,179.386,5.632,149.178
C08011=1189.983,-74.492,-40.795,179.389,5.633,149.177
C08012=1189.977,-74.242,-40.805,179.391,5.634,149.176
C08013=1189.972,-73.992,-40.816,179.393,5.633,149.176
C08014=1189.967,-73.743,-40.827,179.395,5.634,149.175
C08015=1189.962,-73.493,-40.837,179.398,5.634,149.175
C08016=1189.956,-73.244,-40.849,179.400,5.634,149.174
C08017=1189.951,-72.993,-40.859,179.403,5.635,149.173
C08018=1189.946,-72.744,-40.871,179.404,5.635,149.173
C08019=1189.940,-72.494,-40.881,179.407,5.635,149.172
C08020=1189.936,-72.244,-40.892,179.410,5.635,149.171
C08021=1189.929,-71.995,-40.903,179.411,5.635,149.171
C08022=1189.925,-71.745,-40.914,179.414,5.636,149.170
C08023=1189.920,-71.495,-40.925,179.417,5.636,149.169
C08024=1189.914,-71.246,-40.936,179.419,5.636,149.169
C08025=1189.909,-70.996,-40.946,179.421,5.637,149.168
C08026=1189.903,-70.746,-40.958,179.423,5.636,149.167
C08027=1189.898,-70.496,-40.968,179.426,5.637,149.167
C08028=1189.894,-70.246,-40.980,179.428,5.638,149.166
C08029=1189.888,-69.997,-40.990,179.430,5.637,149.166
C08030=1189.883,-69.747,-41.001,179.433,5.638,149.165
C08031=1189.877,-69.497,-41.012,179.435,5.638,149.164
C08032=1189.872,-69.248,-41.023,179.437,5.638,149.164
C08033=1189.867,-68.998,-41.034,179.440,5.638,149.163
C08034=1189.862,-68.749,-41.045,179.442,5.639,149.162
C08035=1189.857,-68.499,-41.057,179.444,5.639,149.162
C08036=1189.852,-68.248,-41.067,179.447,5.639,149.161
C08037=1189.846,-68.000,-41.078,179.449,5.640,149.160
C08038=1189.841,-67.749,-41.089,179.451,5.640,149.160
C08039=1189.835,-67.500,-41.100,179.454,5.640,149.159
C08040=1189.831,-67.250,-41.112,179.456,5.640,149.158
C08041=1189.826,-67.000,-41.122,179.458,5.640,149.158
C08042=1189.820,-66.751,-41.134,179.460,5.641,149.157
C08043=1189.815,-66.501,-41.145,179.463,5.641,149.157
C08044=1189.810,-66.251,-41.155,179.465,5.641,149.156
C08045=1189.805,-66.002,-41.166,179.467,5.642,149.155
C08046=1189.799,-65.752,-41.178,179.469,5.641,149.155
C08047=1189.794,-65.502,-41.189,179.472,5.642,149.154
C08048=1189.789,-65.253,-41.200,179.475,5.642,149.153
C08049=1189.783,-65.003,-41.212,179.476,5.642,149.153
C08050=1189.778,-64.753,-41.222,179.479,5.643,149.152
C08051=1189.773,-64.504,-41.233,179.482,5.643,149.151
C08052=1189.768,-64.254,-41.245,179.484,5.643,149.151
C08053=1189.763,-64.004,-41.256,179.486,5.644,149.150
C08054=1189.758,-63.754,-41.267,179.489,5.644,149.149
C08055=1189.752,-63.505,-41.278,179.491,5.644,149.149
C08056=1189.747,-63.255,-41.290,179.493,5.644,149.148
C08057=1189.742,-63.005,-41.301,179.496,5.645,149.148
C08058=1189.736,-62.756,-41.312,179.498,5.645,149.147
C08059=1189.732,-62.506,-41.323,179.500,5.645,149.146
C08060=1189.726,-62.256,-41.335,179.503,5.646,149.146
C08061=1189.721,-62.006,-41.346,179.505,5.645,149.145
C08062=1189.716,-61.757,-41.357,179.507,5.646,149.144
C08063=1189.710,-61.507,-41.368,179.509,5.647,149.144
C08064=1189.706,-61.258,-41.380,179.512,5.646,149.143
C08065=1189.700,-61.008,-41.392,179.514,5.647,149.142
C08066=1189.695,-60.758,-41.402,179.517,5.647,149.142
C08067=1189.690,-60.508,-41.413,179.518,5.647,149.141
C08068=1189.685,-60.258,-41.425,179.521,5.648,149.141
C08069=1189.680,-60.009,-41.436,179.524,5.648,149.140
C08070=1189.674,-59.760,-41.448,179.526,5.648,149.139
C08071=1189.669,-59.510,-41.459,179.528,5.648,149.139
C08072=1189.664,-59.260,-41.471,179.531,5.649,149.138
C08073=1189.659,-59.010,-41.482,179.533,5.649,149.137
C08074=1189.653,-58.761,-41.492,179.535,5.649,149.137
C08075=1189.648,-58.511,-41.504,179.538,5.650,149.136
C08076=1189.643,-58.261,-41.516,179.540,5.649,149.135
C08077=1189.638,-58.011,-41.528,179.542,5.650,149.135
C08078=1189.633,-57.762,-41.539,179.545,5.651,149.134
C08079=1189.627,-57.513,-41.550,179.547,5.650,149.133
C08080=1189.623,-57.263,-41.562,179.549,5.651,149.133
C08081=1189.617,-57.013,-41.573,179.552,5.651,149.132
C08082=1189.612,-56.763,-41.584,179.554,5.652,149.132
C08083=1189.607,-56.513,-41.596,179.556,5.652,149.131
C08084=1189.601,-56.264,-41.607,179.559,5.652,149.130
C08085=1189.596,-56.014,-41.619,179.562,5.652,149.129
C08086=1189.591,-55.764,-41.630,179.563,5.652,149.129
C08087=1189.586,-55.514,-41.642,179.566,5.653,149.128
C08088=1189.581,-55.265,-41.653,179.569,5.653,149.128
C08089=1189.575,-55.016,-41.665,179.570,5.653,149.127
C08090=1189.570,-54.766,-41.676,179.573,5.654,149.126
C08091=1189.565,-54.516,-41.688,179.575,5.654,149.126
C08092=1189.560,-54.266,-41.699,179.578,5.654,149.125
C08093=1189.555,-54.016,-41.711,179.580,5.655,149.125
C08094=1189.550,-53.767,-41.722,179.582,5.655,149.124
C08095=1189.545,-53.517,-41.734,179.585,5.656,149.123
C08096=1189.539,-53.268,-41.746,179.587,5.655,149.122
C08097=1189.534,-53.018,-41.757,179.589,5.656,149.122
C08098=1189.529,-52.768,-41.769,179.592,5.656,149.121
C08099=1189.524,-52.518,-41.780,179.594,5.656,149.121
C08100=1189.518,-52.268,-41.792,179.597,5.657,149.120
C08101=1189.514,-52.019,-41.804,179.599,5.657,149.119
C08102=1189.509,-51.770,-41.816,179.602,5.658,149.119
C08103=1189.503,-51.520,-41.828,179.604,5.657,149.118
C08104=1189.498,-51.271,-41.839,179.606,5.658,149.117
C08105=1189.492,-51.021,-41.851,179.609,5.659,149.117
C08106=1189.488,-50.771,-41.862,179.611,5.658,149.116
C08107=1189.482,-50.521,-41.874,179.613,5.659,149.115
C08108=1189.477,-50.271,-41.886,179.616,5.659,149.115
C08109=1189.472,-50.022,-41.897,179.618,5.660,149.114
C08110=1189.466,-49.752,-41.910,179.620,5.660,149.113
C08111=1189.461,-49.482,-41.923,179.623,5.660,149.113
C08112=1189.456,-49.211,-41.936,179.626,5.661,149.112
C08113=1189.450,-48.942,-41.948,179.628,5.661,149.111
C08114=1189.444,-48.692,-41.960,179.631,5.661,149.111
C08115=1189.439,-48.442,-41.972,179.633,5.661,149.110
C08116=1189.434,-48.192,-41.984,179.635,5.662,149.109
C08117=1189.429,-47.942,-41.995,179.638,5.662,149.109
C08118=1189.423,-47.692,-42.007,179.640,5.663,149.108
C08119=1189.418,-47.443,-42.020,179.643,5.662,149.107
C08120=1189.414,-47.193,-42.031,179.645,5.663,149.107
C08121=1189.408,-46.943,-42.043,179.647,5.664,149.106
C08122=1189.403,-46.693,-42.055,179.649,5.663,149.105
C08123=1189.398,-46.445,-42.066,179.652,5.664,149.105
C08124=1189.392,-46.195,-42.078,179.654,5.665,149.104
C08125=1189.387,-45.945,-42.090,179.657,5.665,149.104
C08126=1189.381,-45.695,-42.102,179.659,5.665,149.103
C08127=1189.377,-45.446,-42.114,179.662,5.665,149.102
C08128=1189.372,-45.196,-42.126,179.664,5.666,149.102
C08129=1189.366,-44.946,-42.138,179.667,5.666,149.101
C08130=1189.361,-44.696,-42.150,179.669,5.666,149.100
C08131=1189.356,-44.447,-42.162,179.671,5.666,149.100
C08132=1189.351,-44.198,-42.174,179.673,5.667,149.099
C08133=1189.346,-43.948,-42.185,179.676,5.668,149.098
C08134=1189.340,-43.698,-42.198,179.678,5.667,149.098
C08135=1189.336,-43.449,-42.209,179.681,5.668,149.097
C08136=1189.330,-43.199,-42.221,179.683,5.669,149.097
C08137=1189.325,-42.949,-42.234,179.686,5.669,149.096
C08138=1189.320,-42.699,-42.246,179.688,5.669,149.095
C08139=1189.314,-42.450,-42.258,179.690,5.669,149.094
C08140=1189.310,-42.201,-42.270,179.693,5.670,149.094
C08141=1189.304,-41.951,-42.281,179.695,5.670,149.093
C08142=1189.299,-41.701,-42.293,179.697,5.670,149.093
C08143=1189.294,-41.451,-42.306,179.700,5.670,149.092
C08144=1189.288,-41.201,-42.318,179.702,5.671,149.091
C08145=1189.284,-40.952,-42.330,179.705,5.672,149.091
C08146=1189.279,-40.702,-42.342,179.707,5.671,149.090
C08147=1189.273,-40.453,-42.354,179.710,5.672,149.089
C08148=1189.268,-40.203,-42.366,179.712,5.673,149.089
C08149=1189.263,-39.953,-42.378,179.714,5.673,149.088
C08150=1189.258,-39.704,-42.391,179.717,5.673,149.087
C08151=1189.252,-39.454,-42.403,179.719,5.673,149.087
C08152=1189.247,-39.204,-42.414,179.721,5.674,149.086
C08153=1189.242,-38.955,-42.426,179.724,5.674,149.086
C08154=1189.237,-38.705,-42.438,179.726,5.674,149.085
C08155=1189.232,-38.455,-42.451,179.729,5.675,149.084
C08156=1189.227,-38.205,-42.463,179.731,5.675,149.084
C08157=1189.222,-37.956,-42.476,179.734,5.676,149.083
C08158=1189.216,-37.706,-42.488,179.736,5.675,149.082
C08159=1189.211,-37.457,-42.500,179.738,5.676,149.082
C08160=1189.206,-37.207,-42.512,179.741,5.677,149.081
C08161=1189.201,-36.957,-42.525,179.743,5.677,149.080
C08162=1189.196,-36.708,-42.536,179.745,5.677,149.080
C08163=1189.191,-36.458,-42.549,179.748,5.677,149.079
C08164=1189.185,-36.208,-42.561,179.750,5.678,149.079
C08165=1189.180,-35.959,-42.573,179.753,5.679,149.078
C08166=1189.175,-35.710,-42.586,179.755,5.679,149.077
C08167=1189.170,-35.460,-42.598,179.758,5.679,149.076
C08168=1189.165,-35.210,-42.611,179.760,5.680,149.076
C08169=1189.160,-34.960,-42.622,179.762,5.680,149.075
C08170=1189.155,-34.711,-42.635,179.765,5.680,149.075
C08171=1189.149,-34.461,-42.647,179.767,5.680,149.074
C08172=1189.144,-34.211,-42.660,179.770,5.681,149.073
C08173=1189.139,-33.962,-42.672,179.772,5.681,149.073
C08174=1189.134,-33.712,-42.684,179.775,5.682,149.072
C08175=1189.128,-33.463,-42.697,179.777,5.682,149.071
C08176=1189.124,-33.212,-42.709,179.779,5.682,149.071
C08177=1189.119,-32.963,-42.722,179.782,5.683,149.070
C08178=1189.113,-32.714,-42.734,179.784,5.683,149.069
C08179=1189.108,-32.464,-42.746,179.787,5.684,149.069
C08180=1189.103,-32.214,-42.759,179.790,5.684,149.068
C08181=1189.098,-31.965,-42.771,179.791,5.684,149.068
C08182=1189.092,-31.715,-42.783,179.794,5.685,149.067
C08183=1189.088,-31.465,-42.796,179.796,5.685,149.066
C08184=1189.083,-31.216,-42.809,179.799,5.685,149.066
C08185=1189.077,-30.966,-42.821,179.801,5.686,149.065
C08186=1189.072,-30.716,-42.833,179.803,5.686,149.064
C08187=1189.067,-30.467,-42.846,179.806,5.686,149.064
C08188=1189.062,-30.218,-42.858,179.809,5.687,149.063
C08189=1189.057,-29.967,-42.871,179.811,5.688,149.062
C08190=1189.051,-29.718,-42.884,179.813,5.687,149.062
C08191=1189.046,-29.468,-42.896,179.816,5.688,149.061
C08192=1189.041,-29.219,-42.909,179.818,5.688,149.060
C08193=1189.035,-28.969,-42.921,179.820,5.689,149.060
C08194=1189.031,-28.719,-42.934,179.823,5.690,149.059
C08195=1189.026,-28.470,-42.946,179.825,5.689,149.059
C08196=1189.021,-28.220,-42.959,179.828,5.690,149.058
C08197=1189.015,-27.970,-42.971,179.830,5.690,149.057
C08198=1189.010,-27.721,-42.984,179.833,5.691,149.057
C08199=1189.006,-27.471,-42.997,179.835,5.691,149.056
C08200=1189.000,-27.221,-43.010,179.838,5.692,149.055
C08201=1188.995,-26.972,-43.022,179.840,5.692,149.055
C08202=1188.990,-26.723,-43.035,179.842,5.692,149.054
C08203=1188.985,-26.472,-43.047,179.845,5.693,149.053
C08204=1188.980,-26.223,-43.060,179.848,5.693,149.053
C08205=1188.974,-25.973,-43.072,179.850,5.694,149.052
C08206=1188.969,-25.724,-43.085,179.852,5.694,149.052
C08207=1188.964,-25.474,-43.099,179.854,5.694,149.051
C08208=1188.959,-25.225,-43.111,179.857,5.695,149.050
C08209=1188.954,-24.975,-43.124,179.860,5.695,149.049
C08210=1188.948,-24.725,-43.136,179.862,5.696,149.049
C08211=1188.944,-24.475,-43.149,179.865,5.696,149.048
C08212=1188.939,-24.226,-43.161,179.867,5.696,149.048
C08213=1188.933,-23.976,-43.174,179.869,5.697,149.047
C08214=1188.928,-23.707,-43.188,179.872,5.697,149.046
C08215=1188.922,-23.438,-43.201,179.875,5.697,149.045
C08216=1188.917,-23.167,-43.216,179.877,5.698,149.045
C08217=1188.912,-22.898,-43.229,179.880,5.698,149.044
C08218=1188.906,-22.648,-43.243,179.882,5.699,149.044
C08219=1188.901,-22.399,-43.255,179.885,5.700,149.043
C08220=1188.896,-22.149,-43.268,179.887,5.700,149.042
C08221=1188.891,-21.899,-43.281,179.890,5.700,149.042
C08222=1188.885,-21.650,-43.294,179.892,5.701,149.041
C08223=1188.881,-21.400,-43.307,179.894,5.701,149.040
C08224=1188.875,-21.151,-43.319,179.897,5.702,149.040
C08225=1188.870,-20.901,-43.332,179.900,5.702,149.039
C08226=1188.864,-20.652,-43.345,179.902,5.703,149.039
C08227=1188.860,-20.402,-43.358,179.904,5.703,149.038
C08228=1188.855,-20.152,-43.371,179.907,5.703,149.037
C08229=1188.849,-19.903,-43.384,179.909,5.703,149.036
C08230=1188.844,-19.653,-43.397,179.911,5.704,149.036
C08231=1188.839,-19.403,-43.410,179.914,5.705,149.035
C08232=1188.833,-19.154,-43.423,179.917,5.705,149.035
C08233=1188.829,-18.904,-43.436,179.919,5.706,149.034
C08234=1188.824,-18.654,-43.448,179.921,5.706,149.033
C08235=1188.818,-18.405,-43.462,179.924,5.706,149.033
C08236=1188.814,-18.155,-43.475,179.926,5.707,149.032
C08237=1188.809,-17.906,-43.488,179.929,5.707,149.031
C08238=1188.803,-17.656,-43.501,179.931,5.708,149.031
C08239=1188.798,-17.406,-43.514,179.934,5.708,149.030
C08240=1188.793,-17.157,-43.527,179.936,5.708,149.029
C08241=1188.788,-16.907,-43.540,179.939,5.709,149.029
C08242=1188.783,-16.657,-43.553,179.941,5.709,149.028
C08243=1188.778,-16.408,-43.565,179.943,5.710,149.028
C08244=1188.773,-16.158,-43.580,179.946,5.710,149.027
C08245=1188.767,-15.909,-43.592,179.949,5.711,149.026
C08246=1188.763,-15.659,-43.605,179.951,5.711,149.026
C08247=1188.757,-15.409,-43.618,179.954,5.712,149.025
C08248=1188.752,-15.160,-43.631,179.956,5.712,149.024
C08249=1188.747,-14.910,-43.645,179.958,5.712,149.024
C08250=1188.742,-14.661,-43.658,179.961,5.713,149.023
C08251=1188.737,-14.411,-43.671,179.963,5.714,149.023
C08252=1188.731,-14.161,-43.684,179.966,5.714,149.022
C08253=1188.726,-13.912,-43.697,179.968,5.714,149.021
C08254=1188.721,-13.662,-43.711,179.971,5.715,149.020
C08255=1188.716,-13.413,-43.724,179.973,5.715,149.020
C08256=1188.711,-13.163,-43.737,179.975,5.715,149.019
C08257=1188.706,-12.913,-43.750,179.978,5.716,149.019
C08258=1188.701,-12.664,-43.764,179.981,5.716,149.018
C08259=1188.696,-12.414,-43.777,179.983,5.717,149.017
C08260=1188.691,-12.165,-43.789,179.985,5.718,149.017
C08261=1188.686,-11.915,-43.803,179.988,5.718,149.016
C08262=1188.681,-11.666,-43.816,179.991,5.719,149.015
C08263=1188.675,-11.416,-43.830,179.993,5.719,149.015
C08264=1188.670,-11.166,-43.842,179.995,5.719,149.014
C08265=1188.665,-10.917,-43.856,179.998,5.720,149.014
C08266=1188.660,-10.667,-43.869,-180.000,5.720,149.013
C08267=1188.655,-10.417,-43.883,-179.998,5.721,149.012
C08268=1188.650,-10.168,-43.896,-179.995,5.721,149.012
C08269=1188.645,-9.918,-43.909,-179.992,5.722,149.011
C08270=1188.640,-9.669,-43.923,-179.990,5.722,149.010
C08271=1188.635,-9.419,-43.936,-179.987,5.723,149.010
C08272=1188.630,-9.170,-43.949,-179.985,5.724,149.009
C08273=1188.625,-8.920,-43.963,-179.983,5.723,149.008
C08274=1188.620,-8.671,-43.976,-179.980,5.724,149.008
C08275=1188.615,-8.421,-43.990,-179.978,5.725,149.007
C08276=1188.609,-8.171,-44.003,-179.975,5.725,149.007
C08277=1188.604,-7.921,-44.016,-179.973,5.726,149.006
C08278=1188.599,-7.672,-44.030,-179.970,5.726,149.005
C08279=1188.594,-7.422,-44.043,-179.968,5.727,149.005
C08280=1188.589,-7.173,-44.057,-179.965,5.727,149.004
C08281=1188.584,-6.923,-44.070,-179.962,5.728,149.003
C08282=1188.578,-6.674,-44.084,-179.960,5.728,149.003
C08283=1188.573,-6.424,-44.098,-179.958,5.728,149.002
C08284=1188.568,-6.175,-44.111,-179.955,5.729,149.002
C08285=1188.563,-5.925,-44.124,-179.953,5.729,149.001
C08286=1188.558,-5.676,-44.138,-179.950,5.730,149.000
C08287=1188.553,-5.426,-44.151,-179.948,5.731,149.000
C08288=1188.548,-5.177,-44.165,-179.945,5.731,148.999
C08289=1188.543,-4.927,-44.178,-179.943,5.732,148.998
C08290=1188.538,-4.677,-44.192,-179.940,5.732,148.998
C08291=1188.532,-4.427,-44.206,-179.938,5.733,148.997
C08292=1188.528,-4.178,-44.219,-179.935,5.733,148.996
C08293=1188.522,-3.928,-44.233,-179.933,5.734,148.996
C08294=1188.518,-3.679,-44.246,-179.930,5.733,148.995
C08295=1188.512,-3.429,-44.259,-179.928,5.734,148.995
C08296=1188.507,-3.180,-44.274,-179.926,5.735,148.994
C08297=1188.503,-2.930,-44.287,-179.923,5.735,148.993
C08298=1188.497,-2.681,-44.301,-179.920,5.736,148.993
C08299=1188.492,-2.431,-44.315,-179.918,5.737,148.992
C08300=1188.486,-2.181,-44.328,-179.916,5.737,148.991
C08301=1188.482,-1.932,-44.342,-179.913,5.738,148.991
C08302=1188.477,-1.682,-44.356,-179.910,5.738,148.990
C08303=1188.471,-1.433,-44.369,-179.908,5.739,148.990
C08304=1188.467,-1.183,-44.383,-179.905,5.739,148.989
C08305=1188.461,-0.934,-44.396,-179.903,5.740,148.988
C08306=1188.456,-0.684,-44.410,-179.900,5.740,148.987
C08307=1188.451,-0.434,-44.425,-179.898,5.741,148.987
C08308=1188.446,-0.185,-44.437,-179.896,5.741,148.986
C08309=1188.441,0.065,-44.451,-179.893,5.741,148.986
C08310=1188.436,0.315,-44.466,-179.891,5.742,148.985
C08311=1188.430,0.564,-44.479,-179.888,5.743,148.985
C08312=1188.426,0.814,-44.493,-179.886,5.743,148.984
C08313=1188.420,1.063,-44.507,-179.883,5.744,148.983
C08314=1188.416,1.312,-44.521,-179.880,5.744,148.982
C08315=1188.410,1.563,-44.534,-179.878,5.745,148.982
C08316=1188.405,1.811,-44.548,-179.876,5.745,148.981
C08317=1188.400,2.061,-44.562,-179.873,5.746,148.981
C08318=1188.395,2.331,-44.577,-179.870,5.746,148.980
C08319=1188.390,2.600,-44.592,-179.868,5.747,148.979
C08320=1188.384,2.869,-44.607,-179.865,5.747,148.979
C08321=1188.378,3.138,-44.622,-179.862,5.748,148.978
C08322=1188.373,3.388,-44.636,-179.860,5.749,148.977
C08323=1188.368,3.638,-44.650,-179.857,5.749,148.977
C08324=1188.363,3.886,-44.663,-179.855,5.750,148.976
C08325=1188.358,4.137,-44.677,-179.852,5.750,148.975
C08326=1188.353,4.386,-44.691,-179.850,5.751,148.975
C08327=1188.348,4.635,-44.705,-179.847,5.751,148.974
C08328=1188.343,4.885,-44.719,-179.845,5.752,148.974
C08329=1188.338,5.135,-44.734,-179.842,5.752,148.973
C08330=1188.332,5.384,-44.748,-179.840,5.753,148.972
C08331=1188.328,5.633,-44.761,-179.837,5.754,148.972
C08332=1188.323,5.883,-44.775,-179.835,5.754,148.971
C08333=1188.318,6.133,-44.789,-179.832,5.755,148.970
C08334=1188.312,6.382,-44.803,-179.830,5.756,148.970
C08335=1188.307,6.632,-44.817,-179.827,5.756,148.969
C08336=1188.302,6.882,-44.832,-179.824,5.757,148.968
C08337=1188.297,7.131,-44.846,-179.822,5.757,148.968
C08338=1188.292,7.380,-44.860,-179.820,5.758,148.967
C08339=1188.287,7.630,-44.874,-179.817,5.758,148.967
C08340=1188.283,7.879,-44.888,-179.814,5.759,148.966
C08341=1188.278,8.129,-44.902,-179.812,5.759,148.965
C08342=1188.272,8.378,-44.916,-179.810,5.760,148.965
C08343=1188.267,8.628,-44.930,-179.807,5.761,148.964
C08344=1188.262,8.878,-44.944,-179.804,5.761,148.963
C08345=1188.257,9.128,-44.958,-179.802,5.762,148.963
C08346=1188.251,9.377,-44.972,-179.799,5.763,148.962
C08347=1188.246,9.627,-44.986,-179.797,5.763,148.962
C08348=1188.241,9.876,-45.001,-179.794,5.764,148.961
C08349=1188.237,10.126,-45.015,-179.792,5.764,148.960
C08350=1188.232,10.376,-45.029,-179.789,5.765,148.960
C08351=1188.226,10.624,-45.044,-179.787,5.765,148.959
C08352=1188.221,10.874,-45.058,-179.784,5.766,148.958
C08353=1188.216,11.124,-45.072,-179.782,5.767,148.958
C08354=1188.211,11.373,-45.087,-179.779,5.767,148.957
C08355=1188.206,11.623,-45.101,-179.777,5.768,148.957
C08356=1188.201,11.872,-45.115,-179.774,5.768,148.956
C08357=1188.196,12.122,-45.129,-179.772,5.769,148.955
C08358=1188.191,12.371,-45.143,-179.769,5.770,148.955
C08359=1188.186,12.621,-45.158,-179.766,5.770,148.954
C08360=1188.181,12.871,-45.172,-179.764,5.771,148.954
C08361=1188.176,13.120,-45.186,-179.762,5.771,148.953
C08362=1188.171,13.370,-45.200,-179.759,5.772,148.952
C08363=1188.166,13.619,-45.214,-179.756,5.772,148.952
C08364=1188.161,13.868,-45.229,-179.754,5.773,148.951
C08365=1188.156,14.118,-45.244,-179.751,5.774,148.950
C08366=1188.150,14.368,-45.258,-179.749,5.774,148.950
C08367=1188.145,14.618,-45.273,-179.746,5.775,148.949
C08368=1188.140,14.867,-45.287,-179.744,5.776,148.949
C08369=1188.135,15.116,-45.301,-179.741,5.776,148.948
C08370=1188.130,15.366,-45.316,-179.739,5.776,148.947
C08371=1188.125,15.615,-45.330,-179.737,5.777,148.947
C08372=1188.120,15.865,-45.345,-179.734,5.778,148.946
C08373=1188.115,16.115,-45.359,-179.731,5.778,148.945
C08374=1188.110,16.364,-45.373,-179.729,5.779,148.945
C08375=1188.105,16.613,-45.388,-179.726,5.780,148.944
C08376=1188.099,16.863,-45.403,-179.724,5.780,148.944
C08377=1188.095,17.113,-45.417,-179.721,5.781,148.943
C08378=1188.090,17.362,-45.431,-179.719,5.782,148.942
C08379=1188.085,17.611,-45.446,-179.716,5.782,148.942
C08380=1188.080,17.861,-45.460,-179.714,5.783,148.941
C08381=1188.075,18.111,-45.475,-179.711,5.783,148.940
C08382=1188.069,18.361,-45.490,-179.709,5.784,148.940
C08383=1188.065,18.610,-45.505,-179.706,5.784,148.939
C08384=1188.060,18.860,-45.519,-179.704,5.785,148.939
C08385=1188.055,19.109,-45.533,-179.701,5.785,148.938
C08386=1188.050,19.358,-45.548,-179.699,5.786,148.937
C08387=1188.045,19.607,-45.562,-179.696,5.787,148.937
C08388=1188.039,19.857,-45.577,-179.693,5.787,148.936
C08389=1188.034,20.106,-45.592,-179.691,5.788,148.936
C08390=1188.029,20.356,-45.606,-179.689,5.789,148.935
C08391=1188.024,20.606,-45.620,-179.686,5.789,148.934
C08392=1188.019,20.855,-45.636,-179.683,5.790,148.934
C08393=1188.014,21.105,-45.650,-179.681,5.790,148.933
C08394=1188.009,21.354,-45.665,-179.679,5.791,148.932
C08395=1188.004,21.604,-45.680,-179.675,5.792,148.932
C08396=1187.999,21.854,-45.694,-179.673,5.793,148.931
C08397=1187.994,22.103,-45.709,-179.671,5.794,148.931
C08398=1187.989,22.353,-45.724,-179.668,5.794,148.930
C08399=1187.984,22.602,-45.739,-179.665,5.795,148.929
C08400=1187.979,22.852,-45.754,-179.663,5.795,148.929
C08401=1187.974,23.101,-45.769,-179.660,5.796,148.928
C08402=1187.969,23.351,-45.783,-179.658,5.796,148.927
C08403=1187.964,23.600,-45.797,-179.656,5.797,148.927
C08404=1187.959,23.850,-45.813,-179.653,5.798,148.926
C08405=1187.954,24.099,-45.827,-179.650,5.798,148.926
C08406=1187.949,24.348,-45.842,-179.648,5.799,148.925
C08407=1187.943,24.599,-45.857,-179.646,5.800,148.925
C08408=1187.939,24.848,-45.872,-179.643,5.800,148.924
C08409=1187.934,25.097,-45.886,-179.640,5.801,148.923
C08410=1187.928,25.347,-45.902,-179.638,5.802,148.923
C08411=1187.924,25.596,-45.916,-179.635,5.802,148.922
C08412=1187.919,25.846,-45.931,-179.632,5.803,148.921
C08413=1187.913,26.095,-45.947,-179.630,5.804,148.921
C08414=1187.909,26.345,-45.961,-179.627,5.805,148.920
C08415=1187.904,26.594,-45.976,-179.625,5.805,148.920
C08416=1187.898,26.844,-45.991,-179.623,5.806,148.919
C08417=1187.894,27.093,-46.006,-179.620,5.807,148.918
C08418=1187.888,27.343,-46.021,-179.617,5.807,148.918
C08419=1187.883,27.592,-46.036,-179.615,5.808,148.917
C08420=1187.879,27.841,-46.051,-179.612,5.808,148.917
C08421=1187.873,28.091,-46.065,-179.610,5.809,148.916
C08422=1187.868,28.360,-46.081,-179.607,5.810,148.915
C08423=1187.862,28.628,-46.098,-179.604,5.811,148.915
C08424=1187.857,28.897,-46.114,-179.601,5.811,148.914
C08425=1187.851,29.166,-46.130,-179.599,5.812,148.913
C08426=1187.847,29.416,-46.145,-179.597,5.813,148.913
C08427=1187.842,29.665,-46.161,-179.594,5.813,148.912
C08428=1187.837,29.915,-46.175,-179.591,5.814,148.911
C08429=1187.831,30.165,-46.191,-179.588,5.815,148.911
C08430=1187.827,30.414,-46.206,-179.586,5.816,148.910
C08431=1187.822,30.663,-46.220,-179.583,5.816,148.910
C08432=1187.816,30.913,-46.236,-179.581,5.817,148.909
C08433=1187.812,31.162,-46.251,-179.578,5.818,148.909
C08434=1187.806,31.411,-46.266,-179.576,5.818,148.908
C08435=1187.802,31.662,-46.281,-179.573,5.819,148.907
C08436=1187.797,31.911,-46.297,-179.571,5.820,148.907
C08437=1187.792,32.160,-46.312,-179.568,5.820,148.906
C08438=1187.787,32.410,-46.327,-179.565,5.821,148.905
C08439=1187.782,32.659,-46.341,-179.563,5.822,148.905
C08440=1187.776,32.909,-46.357,-179.560,5.823,148.904
C08441=1187.772,33.158,-46.372,-179.558,5.823,148.904
C08442=1187.766,33.407,-46.388,-179.555,5.824,148.903
C08443=1187.761,33.658,-46.403,-179.553,5.825,148.902
C08444=1187.756,33.907,-46.418,-179.550,5.825,148.902
C08445=1187.751,34.156,-46.433,-179.548,5.826,148.901
C08446=1187.746,34.405,-46.448,-179.545,5.827,148.901
C08447=1187.741,34.655,-46.464,-179.542,5.828,148.900
C08448=1187.736,34.904,-46.479,-179.540,5.829,148.900
C08449=1187.732,35.154,-46.495,-179.537,5.829,148.899
C08450=1187.727,35.404,-46.509,-179.535,5.830,148.898
C08451=1187.721,35.653,-46.525,-179.533,5.831,148.898
C08452=1187.716,35.903,-46.540,-179.530,5.831,148.897
C08453=1187.711,36.152,-46.555,-179.527,5.832,148.896
C08454=1187.706,36.402,-46.571,-179.525,5.832,148.896
C08455=1187.702,36.651,-46.586,-179.522,5.834,148.895
C08456=1187.696,36.900,-46.602,-179.519,5.834,148.895
C08457=1187.691,37.150,-46.618,-179.517,5.835,148.894
C08458=1187.686,37.399,-46.633,-179.514,5.836,148.893
C08459=1187.682,37.649,-46.648,-179.512,5.836,148.893
C08460=1187.676,37.898,-46.664,-179.509,5.837,148.892
C08461=1187.672,38.147,-46.679,-179.507,5.838,148.892
C08462=1187.666,38.397,-46.694,-179.504,5.839,148.891
C08463=1187.661,38.647,-46.710,-179.501,5.840,148.890
C08464=1187.656,38.897,-46.725,-179.499,5.840,148.890
C08465=1187.651,39.146,-46.740,-179.496,5.841,148.889
C08466=1187.646,39.395,-46.756,-179.494,5.841,148.889
C08467=1187.641,39.644,-46.771,-179.492,5.842,148.888
C08468=1187.637,39.894,-46.788,-179.489,5.843,148.887
C08469=1187.631,40.143,-46.803,-179.486,5.844,148.887
C08470=1187.627,40.392,-46.818,-179.484,5.845,148.886
C08471=1187.622,40.643,-46.834,-179.481,5.846,148.886
C08472=1187.616,40.892,-46.850,-179.478,5.846,148.885
C08473=1187.611,41.141,-46.865,-179.476,5.847,148.884
C08474=1187.606,41.390,-46.880,-179.473,5.847,148.884
C08475=1187.602,41.641,-46.896,-179.471,5.848,148.883
C08476=1187.596,41.890,-46.912,-179.468,5.850,148.883
C08477=1187.591,42.139,-46.928,-179.465,5.850,148.882
C08478=1187.586,42.388,-46.943,-179.463,5.851,148.881
C08479=1187.581,42.639,-46.959,-179.461,5.852,148.881
C08480=1187.576,42.887,-46.975,-179.458,5.852,148.880
C08481=1187.571,43.137,-46.990,-179.455,5.853,148.880
C08482=1187.567,43.387,-47.006,-179.453,5.854,148.879
C08483=1187.561,43.636,-47.021,-179.450,5.855,148.878
C08484=1187.556,43.885,-47.037,-179.447,5.855,148.878
C08485=1187.551,44.135,-47.053,-179.445,5.856,148.877
C08486=1187.546,44.384,-47.069,-179.443,5.857,148.877
C08487=1187.542,44.633,-47.084,-179.440,5.858,148.876
C08488=1187.537,44.883,-47.100,-179.437,5.859,148.876
C08489=1187.531,45.133,-47.116,-179.435,5.859,148.875
C08490=1187.526,45.382,-47.131,-179.432,5.860,148.874
C08491=1187.521,45.632,-47.148,-179.430,5.861,148.874
C08492=1187.516,45.881,-47.164,-179.427,5.861,148.873
C08493=1187.511,46.130,-47.179,-179.424,5.863,148.873
C08494=1187.507,46.380,-47.195,-179.422,5.864,148.872
C08495=1187.502,46.629,-47.211,-179.419,5.864,148.871
C08496=1187.496,46.878,-47.226,-179.417,5.865,148.871
C08497=1187.491,47.129,-47.242,-179.414,5.865,148.870
C08498=1187.486,47.378,-47.258,-179.412,5.866,148.870
C08499=1187.482,47.627,-47.275,-179.409,5.868,148.869
C08500=1187.477,47.877,-47.290,-179.406,5.868,148.868
C08501=1187.471,48.126,-47.305,-179.404,5.869,148.868
C08502=1187.467,48.375,-47.322,-179.401,5.870,148.867
C08503=1187.462,48.625,-47.337,-179.399,5.870,148.867
C08504=1187.457,48.875,-47.353,-179.396,5.872,148.866
C08505=1187.452,49.124,-47.370,-179.393,5.872,148.866
C08506=1187.446,49.373,-47.385,-179.391,5.873,148.865
C08507=1187.442,49.623,-47.401,-179.389,5.874,148.864
C08508=1187.436,49.872,-47.418,-179.386,5.874,148.864
C08509=1187.432,50.122,-47.434,-179.383,5.876,148.863
C08510=1187.427,50.371,-47.450,-179.381,5.876,148.863
C08511=1187.422,50.621,-47.466,-179.378,5.877,148.862
C08512=1187.416,50.870,-47.481,-179.375,5.877,148.861
C08513=1187.412,51.119,-47.497,-179.373,5.879,148.861
C08514=1187.407,51.369,-47.513,-179.370,5.880,148.860
C08515=1187.402,51.618,-47.529,-179.368,5.881,148.860
C08516=1187.397,51.868,-47.545,-179.365,5.881,148.859
C08517=1187.392,52.117,-47.562,-179.363,5.882,148.858
C08518=1187.388,52.367,-47.578,-179.360,5.883,148.858
C08519=1187.383,52.616,-47.594,-179.357,5.884,148.857
C08520=1187.378,52.866,-47.610,-179.355,5.884,148.857
C08521=1187.373,53.114,-47.626,-179.352,5.885,148.856
C08522=1187.368,53.365,-47.642,-179.350,5.886,148.856
C08523=1187.363,53.613,-47.658,-179.347,5.887,148.855
C08524=1187.357,53.864,-47.675,-179.344,5.888,148.854
C08525=1187.352,54.113,-47.691,-179.342,5.889,148.854
C08526=1187.347,54.381,-47.708,-179.339,5.890,148.853
C08527=1187.342,54.650,-47.726,-179.336,5.891,148.853
C08528=1187.336,54.918,-47.743,-179.334,5.891,148.852
C08529=1187.331,55.187,-47.760,-179.331,5.893,148.851
C08530=1187.326,55.436,-47.777,-179.328,5.893,148.851
C08531=1187.321,55.685,-47.793,-179.326,5.894,148.850
C08532=1187.317,55.935,-47.809,-179.323,5.895,148.850
C08533=1187.311,56.184,-47.825,-179.320,5.896,148.849
C08534=1187.306,56.434,-47.842,-179.318,5.897,148.848
C08535=1187.301,56.683,-47.858,-179.315,5.897,148.848
C08536=1187.296,56.933,-47.874,-179.313,5.898,148.847
C08537=1187.291,57.182,-47.891,-179.310,5.899,148.847
C08538=1187.286,57.431,-47.907,-179.307,5.900,148.846
C08539=1187.282,57.681,-47.923,-179.305,5.901,148.846
C08540=1187.277,57.930,-47.940,-179.302,5.901,148.845
C08541=1187.272,58.180,-47.956,-179.300,5.903,148.844
C08542=1187.266,58.429,-47.972,-179.297,5.904,148.844
C08543=1187.262,58.679,-47.989,-179.294,5.904,148.843
C08544=1187.256,58.928,-48.005,-179.292,5.905,148.843
C08545=1187.252,59.178,-48.021,-179.289,5.906,148.842
C08546=1187.247,59.426,-48.038,-179.287,5.907,148.842
C08547=1187.242,59.676,-48.054,-179.284,5.908,148.841
C08548=1187.237,59.926,-48.072,-179.281,5.909,148.840
C08549=1187.231,60.175,-48.087,-179.279,5.910,148.840
C08550=1187.227,60.425,-48.104,-179.276,5.911,148.839
C08551=1187.222,60.673,-48.120,-179.274,5.911,148.839
C08552=1187.217,60.923,-48.137,-179.271,5.913,148.838
C08553=1187.212,61.173,-48.154,-179.268,5.913,148.837
C08554=1187.207,61.422,-48.170,-179.266,5.914,148.837
C08555=1187.202,61.672,-48.186,-179.263,5.915,148.836
C08556=1187.197,61.920,-48.203,-179.261,5.916,148.836
C08557=1187.192,62.170,-48.220,-179.258,5.917,148.835
C08558=1187.188,62.420,-48.237,-179.255,5.918,148.835
C08559=1187.182,62.669,-48.252,-179.253,5.919,148.834
C08560=1187.178,62.919,-48.269,-179.250,5.920,148.833
C08561=1187.172,63.168,-48.286,-179.248,5.921,148.833
C08562=1187.167,63.417,-48.302,-179.245,5.921,148.832
C08563=1187.163,63.667,-48.319,-179.242,5.923,148.832
C08564=1187.157,63.916,-48.336,-179.240,5.923,148.831
C08565=1187.153,64.165,-48.353,-179.237,5.924,148.831
C08566=1187.148,64.415,-48.369,-179.235,5.925,148.830
C08567=1187.143,64.663,-48.386,-179.232,5.926,148.830
C08568=1187.138,64.914,-48.402,-179.229,5.927,148.829
C08569=1187.133,65.163,-48.419,-179.227,5.928,148.828
C08570=1187.128,65.412,-48.435,-179.224,5.929,148.828
C08571=1187.123,65.662,-48.452,-179.222,5.930,148.827
C08572=1187.118,65.911,-48.469,-179.219,5.930,148.827
C08573=1187.114,66.161,-48.486,-179.216,5.932,148.826
C08574=1187.108,66.410,-48.503,-179.214,5.933,148.826
C08575=1187.104,66.659,-48.519,-179.211,5.933,148.825
C08576=1187.098,66.909,-48.537,-179.209,5.934,148.824
C08577=1187.093,67.158,-48.553,-179.206,5.935,148.824
C08578=1187.089,67.408,-48.570,-179.204,5.936,148.823
C08579=1187.084,67.657,-48.587,-179.201,5.937,148.823
C08580=1187.078,67.906,-48.603,-179.198,5.939,148.822
C08581=1187.074,68.156,-48.620,-179.196,5.939,148.822
C08582=1187.069,68.405,-48.637,-179.193,5.940,148.821
C08583=1187.065,68.654,-48.654,-179.190,5.941,148.821
C08584=1187.059,68.903,-48.671,-179.188,5.942,148.820
C08585=1187.054,69.153,-48.688,-179.186,5.943,148.819
C08586=1187.049,69.403,-48.705,-179.182,5.944,148.819
C08587=1187.045,69.652,-48.722,-179.180,5.945,148.818
C08588=1187.039,69.901,-48.738,-179.178,5.946,148.818
C08589=1187.034,70.151,-48.756,-179.174,5.947,148.817
C08590=1187.030,70.400,-48.772,-179.172,5.948,148.817
C08591=1187.025,70.650,-48.789,-179.170,5.948,148.816
C08592=1187.020,70.898,-48.806,-179.167,5.950,148.816
C08593=1187.015,71.148,-48.824,-179.164,5.951,148.815
C08594=1187.010,71.397,-48.840,-179.162,5.951,148.814
C08595=1187.005,71.647,-48.858,-179.159,5.953,148.814
C08596=1187.000,71.897,-48.874,-179.157,5.954,148.813
C08597=1186.995,72.146,-48.891,-179.154,5.954,148.813
C08598=1186.990,72.395,-48.909,-179.151,5.956,148.812
C08599=1186.985,72.644,-48.926,-179.149,5.957,148.812
C08600=1186.981,72.894,-48.943,-179.146,5.957,148.811
C08601=1186.975,73.144,-48.960,-179.143,5.959,148.811
C08602=1186.971,73.392,-48.977,-179.141,5.959,148.810
C08603=1186.965,73.642,-48.994,-179.139,5.960,148.809
C08604=1186.961,73.891,-49.011,-179.135,5.962,148.809
C08605=1186.956,74.141,-49.028,-179.133,5.962,148.808
C08606=1186.951,74.390,-49.046,-179.131,5.963,148.808
C08607=1186.946,74.639,-49.062,-179.127,5.964,148.807
C08608=1186.941,74.889,-49.080,-179.125,5.965,148.807
C08609=1186.936,75.138,-49.096,-179.123,5.966,148.806
C08610=1186.931,75.387,-49.114,-179.120,5.968,148.806
C08611=1186.927,75.637,-49.131,-179.117,5.968,148.805
C08612=1186.921,75.887,-49.148,-179.115,5.969,148.804
C08613=1186.916,76.135,-49.166,-179.112,5.970,148.804
C08614=1186.912,76.385,-49.182,-179.110,5.971,148.803
C08615=1186.907,76.634,-49.200,-179.107,5.973,148.803
C08616=1186.901,76.884,-49.218,-179.105,5.973,148.802
C08617=1186.897,77.133,-49.234,-179.102,5.974,148.802
C08618=1186.892,77.382,-49.252,-179.099,5.976,148.801
C08619=1186.888,77.632,-49.269,-179.097,5.976,148.801
C08620=1186.882,77.882,-49.286,-179.094,5.977,148.800
C08621=1186.877,78.130,-49.304,-179.091,5.979,148.799
C08622=1186.872,78.379,-49.321,-179.089,5.979,148.799
C08623=1186.867,78.629,-49.339,-179.086,5.980,148.798
C08624=1186.862,78.878,-49.356,-179.083,5.981,148.798
C08625=1186.858,79.127,-49.373,-179.081,5.982,148.797
C08626=1186.853,79.377,-49.390,-179.078,5.984,148.797
C08627=1186.848,79.626,-49.408,-179.076,5.984,148.796
C08628=1186.843,79.876,-49.426,-179.073,5.985,148.796
C08629=1186.838,80.125,-49.443,-179.070,5.987,148.795
C08630=1186.832,80.393,-49.461,-179.068,5.987,148.794
C08631=1186.827,80.662,-49.480,-179.065,5.989,148.794
C08632=1186.822,80.930,-49.500,-179.062,5.990,148.793
C08633=1186.817,81.199,-49.518,-179.059,5.991,148.793
C08634=1186.812,81.448,-49.536,-179.057,5.991,148.792
C08635=1186.807,81.698,-49.553,-179.054,5.993,148.792
C08636=1186.802,81.947,-49.571,-179.051,5.994,148.791
C08637=1186.797,82.197,-49.588,-179.049,5.995,148.791
C08638=1186.793,82.446,-49.606,-179.046,5.996,148.790
C08639=1186.787,82.694,-49.623,-179.044,5.997,148.790
C08640=1186.782,82.944,-49.640,-179.041,5.998,148.789
C08641=1186.777,83.193,-49.658,-179.038,5.999,148.788
C08642=1186.773,83.443,-49.675,-179.035,6.001,148.788
C08643=1186.768,83.692,-49.693,-179.033,6.001,148.787
C08644=1186.763,83.941,-49.711,-179.030,6.002,148.787
C08645=1186.758,84.191,-49.728,-179.028,6.004,148.786
C08646=1186.753,84.440,-49.746,-179.025,6.004,148.786
C08647=1186.748,84.689,-49.764,-179.022,6.006,148.785
C08648=1186.743,84.939,-49.781,-179.020,6.007,148.785
C08649=1186.739,85.188,-49.799,-179.018,6.007,148.784
C08650=1186.734,85.437,-49.817,-179.014,6.009,148.784
C08651=1186.728,85.687,-49.834,-179.012,6.010,148.783
C08652=1186.724,85.936,-49.852,-179.009,6.011,148.782
C08653=1186.719,86.185,-49.870,-179.007,6.012,148.782
C08654=1186.714,86.434,-49.888,-179.004,6.013,148.781
C08655=1186.710,86.684,-49.905,-179.002,6.014,148.781
C08656=1186.705,86.934,-49.923,-178.999,6.015,148.780
C08657=1186.700,87.183,-49.941,-178.996,6.017,148.780
C08658=1186.695,87.432,-49.959,-178.994,6.017,148.779
C08659=1186.690,87.682,-49.976,-178.991,6.019,148.779
C08660=1186.685,87.931,-49.994,-178.988,6.019,148.778
C08661=1186.680,88.180,-50.012,-178.986,6.021,148.778
C08662=1186.675,88.429,-50.030,-178.983,6.022,148.777
C08663=1186.670,88.678,-50.048,-178.981,6.023,148.777
C08664=1186.665,88.928,-50.066,-178.978,6.024,148.776
C08665=1186.660,89.177,-50.083,-178.975,6.025,148.776
C08666=1186.655,89.427,-50.101,-178.972,6.026,148.775
C08667=1186.650,89.676,-50.119,-178.970,6.027,148.775
C08668=1186.645,89.925,-50.137,-178.967,6.028,148.774
C08669=1186.640,90.174,-50.155,-178.965,6.029,148.773
C08670=1186.636,90.424,-50.174,-178.962,6.031,148.773
C08671=1186.631,90.673,-50.192,-178.959,6.032,148.772
C08672=1186.626,90.922,-50.210,-178.957,6.033,148.772
C08673=1186.621,91.172,-50.227,-178.954,6.034,148.771
C08674=1186.616,91.421,-50.245,-178.952,6.035,148.771
C08675=1186.611,91.670,-50.263,-178.949,6.036,148.770
C08676=1186.606,91.920,-50.281,-178.947,6.037,148.770
C08677=1186.601,92.169,-50.299,-178.943,6.038,148.769
C08678=1186.597,92.418,-50.317,-178.941,6.039,148.769
C08679=1186.592,92.668,-50.335,-178.938,6.041,148.768
C08680=1186.587,92.917,-50.353,-178.936,6.042,148.768
C08681=1186.582,93.166,-50.371,-178.933,6.043,148.767
C08682=1186.577,93.415,-50.389,-178.931,6.044,148.767
C08683=1186.573,93.665,-50.407,-178.927,6.045,148.766
C08684=1186.568,93.914,-50.425,-178.925,6.046,148.766
C08685=1186.563,94.164,-50.443,-178.923,6.047,148.765
C08686=1186.558,94.413,-50.461,-178.920,6.049,148.765
C08687=1186.553,94.662,-50.479,-178.918,6.049,148.764
C08688=1186.549,94.911,-50.497,-178.915,6.051,148.763
C08689=1186.544,95.160,-50.515,-178.913,6.052,148.763
C08690=1186.538,95.409,-50.535,-178.909,6.053,148.762
C08691=1186.534,95.659,-50.553,-178.907,6.054,148.762
C08692=1186.529,95.908,-50.571,-178.904,6.055,148.761
C08693=1186.524,96.157,-50.589,-178.902,6.056,148.761
C08694=1186.519,96.407,-50.607,-178.899,6.058,148.760
C08695=1186.514,96.656,-50.625,-178.897,6.059,148.760
C08696=1186.510,96.906,-50.643,-178.894,6.060,148.759
C08697=1186.504,97.155,-50.662,-178.891,6.061,148.759
C08698=1186.500,97.404,-50.681,-178.888,6.063,148.758
C08699=1186.495,97.653,-50.699,-178.886,6.063,148.758
C08700=1186.490,97.902,-50.716,-178.883,6.065,148.757
C08701=1186.486,98.152,-50.735,-178.881,6.065,148.757
C08702=1186.480,98.401,-50.753,-178.878,6.067,148.756
C08703=1186.475,98.651,-50.771,-178.875,6.068,148.756
C08704=1186.471,98.899,-50.790,-178.872,6.069,148.755
C08705=1186.466,99.149,-50.808,-178.870,6.070,148.755
C08706=1186.461,99.398,-50.826,-178.867,6.072,148.754
C08707=1186.456,99.648,-50.845,-178.865,6.073,148.754
C08708=1186.451,99.896,-50.864,-178.862,6.074,148.753
C08709=1186.447,100.146,-50.882,-178.860,6.075,148.753
C08710=1186.442,100.395,-50.900,-178.856,6.076,148.752
C08711=1186.436,100.645,-50.919,-178.854,6.077,148.752
C08712=1186.432,100.894,-50.938,-178.852,6.079,148.751
C08713=1186.427,101.143,-50.956,-178.849,6.080,148.751
C08714=1186.422,101.392,-50.974,-178.846,6.081,148.750
C08715=1186.417,101.641,-50.993,-178.844,6.082,148.750
C08716=1186.413,101.891,-51.011,-178.841,6.084,148.749
C08717=1186.408,102.140,-51.029,-178.839,6.084,148.749
C08718=1186.402,102.389,-51.049,-178.836,6.086,148.748
C08719=1186.398,102.639,-51.067,-178.834,6.087,148.748
C08720=1186.393,102.888,-51.085,-178.830,6.088,148.747
C08721=1186.388,103.137,-51.104,-178.828,6.089,148.747
C08722=1186.384,103.387,-51.122,-178.825,6.090,148.746
C08723=1186.379,103.636,-51.141,-178.822,6.092,148.746
C08724=1186.373,103.885,-51.160,-178.820,6.093,148.745
C08725=1186.369,104.135,-51.178,-178.817,6.094,148.745
C08726=1186.364,104.383,-51.197,-178.815,6.095,148.744
C08727=1186.359,104.633,-51.215,-178.812,6.097,148.743
C08728=1186.355,104.882,-51.234,-178.810,6.098,148.743
C08729=1186.350,105.131,-51.252,-178.807,6.099,148.743
C08730=1186.344,105.380,-51.272,-178.804,6.100,148.742
C08731=1186.340,105.630,-51.290,-178.801,6.102,148.742
C08732=1186.335,105.879,-51.309,-178.799,6.102,148.741
C08733=1186.330,106.128,-51.327,-178.796,6.104,148.741
C08734=1186.325,106.397,-51.348,-178.793,6.105,148.740
C08735=1186.320,106.665,-51.368,-178.791,6.106,148.739
C08736=1186.314,106.934,-51.388,-178.788,6.108,148.739
C08737=1186.310,107.202,-51.408,-178.785,6.109,148.738
C08738=1186.304,107.451,-51.427,-178.782,6.110,148.738
C08739=1186.300,107.701,-51.446,-178.780,6.112,148.737
C08740=1186.295,107.950,-51.465,-178.777,6.114,148.737
C08741=1186.290,108.199,-51.483,-178.774,6.114,148.736
C08742=1186.285,108.448,-51.503,-178.772,6.116,148.736
C08743=1186.280,108.697,-51.521,-178.769,6.116,148.735
C08744=1186.276,108.947,-51.540,-178.766,6.118,148.735
C08745=1186.271,109.196,-51.559,-178.764,6.119,148.734
C08746=1186.265,109.445,-51.578,-178.761,6.120,148.734
C08747=1186.261,109.694,-51.597,-178.758,6.122,148.733
C08748=1186.256,109.943,-51.616,-178.756,6.123,148.733
C08749=1186.252,110.193,-51.634,-178.753,6.124,148.732
C08750=1186.246,110.442,-51.654,-178.751,6.125,148.732
C08751=1186.242,110.691,-51.673,-178.748,6.127,148.731
C08752=1186.237,110.941,-51.691,-178.745,6.128,148.731
C08753=1186.233,111.190,-51.710,-178.743,6.129,148.731
C08754=1186.227,111.439,-51.730,-178.740,6.131,148.730
C08755=1186.223,111.689,-51.748,-178.737,6.132,148.730
C08756=1186.218,111.938,-51.767,-178.735,6.133,148.729
C08757=1186.212,112.186,-51.787,-178.732,6.134,148.728
C08758=1186.208,112.436,-51.806,-178.729,6.136,148.728
C08759=1186.203,112.685,-51.824,-178.726,6.137,148.727
C08760=1186.199,112.934,-51.843,-178.724,6.138,148.727
C08761=1186.193,113.183,-51.863,-178.721,6.140,148.727
C08762=1186.189,113.433,-51.882,-178.719,6.140,148.726
C08763=1186.184,113.681,-51.901,-178.716,6.142,148.726
C08764=1186.179,113.932,-51.920,-178.713,6.144,148.725
C08765=1186.174,114.180,-51.939,-178.711,6.144,148.725
C08766=1186.170,114.430,-51.958,-178.708,6.146,148.724
C08767=1186.164,114.679,-51.978,-178.706,6.147,148.724
C08768=1186.160,114.928,-51.997,-178.703,6.149,148.723
C08769=1186.155,115.177,-52.016,-178.700,6.150,148.723
C08770=1186.150,115.427,-52.035,-178.698,6.151,148.722
C08771=1186.146,115.676,-52.054,-178.695,6.153,148.722
C08772=1186.140,115.925,-52.073,-178.693,6.154,148.721
C08773=1186.136,116.175,-52.093,-178.690,6.155,148.721
C08774=1186.131,116.423,-52.112,-178.687,6.157,148.720
C08775=1186.126,116.673,-52.131,-178.685,6.158,148.720
C08776=1186.121,116.922,-52.151,-178.682,6.159,148.719
C08777=1186.116,117.171,-52.170,-178.679,6.160,148.719
C08778=1186.112,117.420,-52.189,-178.677,6.162,148.718
C08779=1186.107,117.669,-52.209,-178.674,6.163,148.718
C08780=1186.102,117.919,-52.228,-178.671,6.164,148.717
C08781=1186.098,118.167,-52.247,-178.669,6.166,148.717
C08782=1186.093,118.417,-52.267,-178.666,6.167,148.717
C08783=1186.088,118.666,-52.286,-178.663,6.168,148.716
C08784=1186.083,118.915,-52.305,-178.661,6.170,148.715
C08785=1186.079,119.165,-52.325,-178.658,6.171,148.715
C08786=1186.073,119.414,-52.344,-178.655,6.172,148.714
C08787=1186.069,119.663,-52.363,-178.653,6.174,148.714
C08788=1186.063,119.912,-52.383,-178.650,6.175,148.714
C08789=1186.059,120.162,-52.402,-178.647,6.176,148.713
C08790=1186.055,120.411,-52.422,-178.645,6.178,148.713
C08791=1186.049,120.660,-52.441,-178.642,6.179,148.712
C08792=1186.044,120.909,-52.460,-178.639,6.180,148.712
C08793=1186.040,121.159,-52.480,-178.637,6.182,148.711
C08794=1186.034,121.408,-52.499,-178.634,6.183,148.711
C08795=1186.030,121.657,-52.520,-178.631,6.184,148.710
C08796=1186.025,121.905,-52.538,-178.629,6.186,148.710
C08797=1186.021,122.155,-52.558,-178.626,6.187,148.709
C08798=1186.016,122.404,-52.578,-178.623,6.188,148.709
C08799=1186.011,122.653,-52.597,-178.621,6.189,148.708
C08800=1186.006,122.903,-52.617,-178.618,6.191,148.708
C08801=1186.001,123.152,-52.637,-178.616,6.193,148.708
C08802=1185.996,123.401,-52.656,-178.613,6.193,148.707
C08803=1185.992,123.650,-52.675,-178.610,6.195,148.707
C08804=1185.987,123.899,-52.695,-178.608,6.197,148.706
C08805=1185.983,124.149,-52.715,-178.605,6.197,148.705
C08806=1185.977,124.397,-52.735,-178.602,6.199,148.705
C08807=1185.973,124.647,-52.754,-178.600,6.201,148.705
C08808=1185.968,124.896,-52.774,-178.597,6.202,148.704
C08809=1185.963,125.145,-52.793,-178.594,6.203,148.704
C08810=1185.958,125.394,-52.814,-178.592,6.205,148.703
C08811=1185.953,125.644,-52.833,-178.590,6.206,148.703
C08812=1185.949,125.893,-52.853,-178.586,6.207,148.702
C08813=1185.944,126.142,-52.873,-178.584,6.209,148.702
C08814=1185.939,126.391,-52.893,-178.582,6.210,148.701
C08815=1185.934,126.641,-52.912,-178.578,6.211,148.701
C08816=1185.929,126.889,-52.932,-178.576,6.213,148.700
C08817=1185.924,127.138,-52.952,-178.573,6.215,148.700
C08818=1185.920,127.388,-52.972,-178.571,6.216,148.700
C08819=1185.915,127.637,-52.992,-178.568,6.217,148.699
C08820=1185.911,127.887,-53.012,-178.565,6.219,148.699
C08821=1185.905,128.135,-53.031,-178.563,6.220,148.698
C08822=1185.901,128.384,-53.051,-178.560,6.222,148.698
C08823=1185.896,128.634,-53.071,-178.557,6.223,148.697
C08824=1185.892,128.883,-53.091,-178.555,6.224,148.697
C08825=1185.886,129.132,-53.111,-178.552,6.226,148.696
C08826=1185.882,129.381,-53.131,-178.549,6.227,148.696
C08827=1185.877,129.630,-53.151,-178.547,6.228,148.695
C08828=1185.872,129.880,-53.170,-178.544,6.230,148.695
C08829=1185.868,130.129,-53.191,-178.541,6.232,148.695
C08830=1185.862,130.378,-53.210,-178.538,6.233,148.694
C08831=1185.858,130.627,-53.230,-178.536,6.234,148.694
C08832=1185.853,130.876,-53.250,-178.533,6.236,148.693
C08833=1185.849,131.125,-53.270,-178.531,6.237,148.693
C08834=1185.844,131.375,-53.290,-178.528,6.238,148.692
C08835=1185.838,131.623,-53.311,-178.525,6.240,148.692
C08836=1185.834,131.872,-53.331,-178.523,6.242,148.691
C08837=1185.829,132.122,-53.351,-178.520,6.243,148.691
C08838=1185.824,132.390,-53.372,-178.517,6.245,148.690
C08839=1185.819,132.659,-53.394,-178.515,6.246,148.690
C08840=1185.814,132.927,-53.415,-178.512,6.247,148.689
C08841=1185.809,133.196,-53.438,-178.509,6.249,148.689
C08842=1185.804,133.445,-53.457,-178.506,6.251,148.689
C08843=1185.799,133.694,-53.478,-178.503,6.252,148.688
C08844=1185.795,133.944,-53.497,-178.500,6.254,148.688
C08845=1185.790,134.193,-53.518,-178.498,6.255,148.687
C08846=1185.785,134.442,-53.539,-178.496,6.256,148.687
C08847=1185.780,134.691,-53.558,-178.493,6.258,148.686
C08848=1185.775,134.940,-53.578,-178.490,6.259,148.686
C08849=1185.771,135.189,-53.599,-178.488,6.261,148.685
C08850=1185.765,135.439,-53.619,-178.485,6.262,148.685
C08851=1185.761,135.688,-53.639,-178.482,6.264,148.685
C08852=1185.757,135.937,-53.660,-178.480,6.265,148.684
C08853=1185.752,136.186,-53.680,-178.477,6.266,148.684
C08854=1185.747,136.435,-53.700,-178.474,6.268,148.683
C08855=1185.742,136.684,-53.721,-178.471,6.270,148.683
C08856=1185.738,136.933,-53.741,-178.469,6.271,148.682
C08857=1185.733,137.182,-53.761,-178.466,6.272,148.682
C08858=1185.727,137.431,-53.781,-178.463,6.274,148.681
C08859=1185.723,137.680,-53.802,-178.461,6.276,148.681
C08860=1185.718,137.929,-53.822,-178.459,6.277,148.681
C08861=1185.713,138.179,-53.843,-178.455,6.278,148.680
C08862=1185.709,138.428,-53.863,-178.453,6.280,148.680
C08863=1185.704,138.677,-53.883,-178.450,6.282,148.679
C08864=1185.700,138.926,-53.903,-178.448,6.283,148.679
C08865=1185.694,139.175,-53.924,-178.445,6.284,148.678
C08866=1185.690,139.424,-53.945,-178.442,6.286,148.678
C08867=1185.686,139.673,-53.965,-178.439,6.288,148.677
C08868=1185.680,139.923,-53.986,-178.437,6.289,148.677
C08869=1185.676,140.171,-54.007,-178.435,6.290,148.677
C08870=1185.671,140.421,-54.028,-178.432,6.292,148.676
C08871=1185.666,140.670,-54.047,-178.429,6.293,148.676
C08872=1185.662,140.919,-54.068,-178.426,6.295,148.675
C08873=1185.656,141.168,-54.088,-178.424,6.296,148.675
C08874=1185.652,141.417,-54.109,-178.421,6.298,148.675
C08875=1185.648,141.666,-54.129,-178.419,6.300,148.674
C08876=1185.642,141.916,-54.150,-178.415,6.301,148.674
C08877=1185.638,142.165,-54.171,-178.413,6.303,148.673
C08878=1185.633,142.414,-54.192,-178.411,6.304,148.673
C08879=1185.628,142.663,-54.212,-178.408,6.305,148.672
C08880=1185.623,142.912,-54.233,-178.405,6.307,148.672
C08881=1185.619,143.161,-54.253,-178.402,6.309,148.671
C08882=1185.614,143.410,-54.274,-178.400,6.310,148.671
C08883=1185.609,143.659,-54.295,-178.397,6.311,148.671
C08884=1185.605,143.908,-54.315,-178.395,6.313,148.670
C08885=1185.599,144.157,-54.336,-178.392,6.315,148.670
C08886=1185.595,144.406,-54.356,-178.389,6.317,148.669
C08887=1185.590,144.656,-54.377,-178.387,6.317,148.669
C08888=1185.586,144.905,-54.399,-178.384,6.319,148.668
C08889=1185.581,145.154,-54.420,-178.381,6.321,148.668
C08890=1185.577,145.403,-54.440,-178.378,6.323,148.668
C08891=1185.572,145.652,-54.461,-178.376,6.324,148.667
C08892=1185.567,145.901,-54.481,-178.373,6.326,148.667
C08893=1185.562,146.150,-54.502,-178.371,6.327,148.666
C08894=1185.557,146.399,-54.523,-178.368,6.328,148.666
C08895=1185.553,146.648,-54.544,-178.365,6.330,148.666
C08896=1185.548,146.897,-54.565,-178.362,6.332,148.665
C08897=1185.543,147.146,-54.586,-178.360,6.334,148.665
C08898=1185.538,147.395,-54.607,-178.358,6.335,148.664
C08899=1185.534,147.645,-54.627,-178.354,6.336,148.664
C08900=1185.529,147.894,-54.648,-178.352,6.338,148.663
C08901=1185.525,148.143,-54.670,-178.349,6.340,148.663
C08902=1185.519,148.392,-54.690,-178.346,6.341,148.663
C08903=1185.514,148.641,-54.711,-178.344,6.343,148.662
C08904=1185.510,148.890,-54.732,-178.342,6.344,148.662
C08905=1185.505,149.139,-54.754,-178.339,6.346,148.661
C08906=1185.501,149.388,-54.774,-178.336,6.347,148.661
C08907=1185.496,149.638,-54.795,-178.333,6.349,148.660
C08908=1185.491,149.886,-54.817,-178.330,6.351,148.660
C08909=1185.487,150.135,-54.837,-178.328,6.353,148.660
C08910=1185.482,150.385,-54.858,-178.326,6.354,148.659
C08911=1185.477,150.633,-54.880,-178.323,6.355,148.659
C08912=1185.472,150.882,-54.900,-178.320,6.357,148.659
C08913=1185.468,151.132,-54.922,-178.318,6.359,148.658
C08914=1185.463,151.381,-54.943,-178.314,6.360,148.658
C08915=1185.458,151.630,-54.964,-178.312,6.362,148.657
C08916=1185.453,151.879,-54.985,-178.310,6.363,148.657
C08917=1185.448,152.128,-55.006,-178.307,6.365,148.656
C08918=1185.444,152.377,-55.027,-178.304,6.366,148.656
C08919=1185.440,152.626,-55.049,-178.301,6.368,148.656
C08920=1185.434,152.875,-55.070,-178.299,6.370,148.655
C08921=1185.430,153.124,-55.091,-178.296,6.372,148.655
C08922=1185.425,153.373,-55.112,-178.293,6.373,148.654
C08923=1185.421,153.623,-55.133,-178.291,6.374,148.654
C08924=1185.416,153.871,-55.155,-178.288,6.376,148.654
C08925=1185.410,154.121,-55.176,-178.285,6.378,148.653
C08926=1185.406,154.369,-55.197,-178.283,6.379,148.653
C08927=1185.402,154.619,-55.218,-178.280,6.381,148.652
C08928=1185.397,154.867,-55.240,-178.277,6.383,148.652
C08929=1185.392,155.117,-55.261,-178.275,6.385,148.652
C08930=1185.387,155.365,-55.283,-178.272,6.387,148.651
C08931=1185.383,155.615,-55.303,-178.269,6.387,148.651
C08932=1185.378,155.864,-55.325,-178.267,6.389,148.650
C08933=1185.373,156.112,-55.347,-178.264,6.391,148.650
C08934=1185.368,156.362,-55.368,-178.261,6.392,148.650
C08935=1185.364,156.611,-55.390,-178.259,6.394,148.649
C08936=1185.359,156.860,-55.411,-178.256,6.396,148.649
C08937=1185.355,157.108,-55.432,-178.253,6.398,148.648
C08938=1185.350,157.358,-55.454,-178.251,6.400,148.648
C08939=1185.345,157.607,-55.475,-178.249,6.400,148.648
C08940=1185.340,157.856,-55.496,-178.246,6.402,148.647
C08941=1185.336,158.105,-55.518,-178.243,6.404,148.647
C08942=1185.331,158.373,-55.541,-178.240,6.405,148.646
C08943=1185.325,158.643,-55.564,-178.237,6.408,148.646
C08944=1185.320,158.912,-55.587,-178.234,6.410,148.646
C08945=1185.315,159.181,-55.611,-178.231,6.412,148.645
C08946=1185.311,159.431,-55.632,-178.228,6.413,148.645
C08947=1185.306,159.679,-55.654,-178.226,6.415,148.644
C08948=1185.301,159.928,-55.676,-178.223,6.417,148.644
C08949=1185.297,160.177,-55.698,-178.221,6.418,148.643
C08950=1185.292,160.426,-55.718,-178.218,6.419,148.643
C08951=1185.287,160.675,-55.740,-178.215,6.421,148.643
C08952=1185.283,160.924,-55.762,-178.213,6.423,148.642
C08953=1185.278,161.173,-55.784,-178.210,6.425,148.642
C08954=1185.273,161.421,-55.805,-178.207,6.426,148.642
C08955=1185.269,161.671,-55.827,-178.205,6.428,148.641
C08956=1185.264,161.920,-55.848,-178.202,6.430,148.641
C08957=1185.260,162.169,-55.870,-178.199,6.432,148.641
C08958=1185.255,162.418,-55.892,-178.197,6.433,148.640
C08959=1185.250,162.667,-55.914,-178.194,6.435,148.640
C08960=1185.246,162.916,-55.936,-178.191,6.437,148.639
C08961=1185.240,163.165,-55.957,-178.189,6.438,148.639
C08962=1185.236,163.415,-55.979,-178.186,6.440,148.639
C08963=1185.231,163.663,-56.000,-178.183,6.441,148.638
C08964=1185.226,163.912,-56.022,-178.181,6.443,148.638
C08965=1185.222,164.161,-56.044,-178.178,6.445,148.637
C08966=1185.217,164.410,-56.066,-178.175,6.447,148.637
C08967=1185.212,164.659,-56.088,-178.173,6.448,148.637
C08968=1185.207,164.908,-56.110,-178.170,6.450,148.636
C08969=1185.203,165.157,-56.132,-178.167,6.452,148.636
C08970=1185.198,165.406,-56.154,-178.165,6.454,148.635
C08971=1185.194,165.655,-56.176,-178.162,6.455,148.635
C08972=1185.189,165.904,-56.198,-178.159,6.457,148.635
C08973=1185.184,166.153,-56.219,-178.157,6.459,148.634
C08974=1185.180,166.402,-56.241,-178.154,6.461,148.634
C08975=1185.175,166.651,-56.263,-178.151,6.462,148.634
C08976=1185.170,166.900,-56.286,-178.148,6.464,148.633
C08977=1185.165,167.149,-56.307,-178.146,6.466,148.633
C08978=1185.161,167.398,-56.329,-178.144,6.467,148.632
C08979=1185.156,167.647,-56.351,-178.141,6.469,148.632
C08980=1185.152,167.896,-56.373,-178.138,6.471,148.632
C08981=1185.147,168.145,-56.395,-178.136,6.472,148.631
C08982=1185.142,168.395,-56.417,-178.133,6.474,148.631
C08983=1185.137,168.643,-56.439,-178.130,6.476,148.631
C08984=1185.133,168.892,-56.462,-178.128,6.478,148.630
C08985=1185.128,169.141,-56.484,-178.125,6.479,148.630
C08986=1185.124,169.390,-56.506,-178.122,6.481,148.630
C08987=1185.118,169.639,-56.528,-178.120,6.483,148.629
C08988=1185.114,169.888,-56.550,-178.117,6.485,148.629
C08989=1185.109,170.137,-56.572,-178.114,6.487,148.628
C08990=1185.105,170.386,-56.594,-178.112,6.488,148.628
C08991=1185.100,170.635,-56.617,-178.109,6.490,148.628
C08992=1185.095,170.884,-56.639,-178.106,6.492,148.627
C08993=1185.091,171.133,-56.661,-178.104,6.494,148.627
C08994=1185.086,171.382,-56.682,-178.101,6.495,148.627
C08995=1185.082,171.631,-56.706,-178.098,6.497,148.626
C08996=1185.077,171.880,-56.727,-178.096,6.499,148.626
C08997=1185.072,172.129,-56.750,-178.093,6.501,148.626
C08998=1185.068,172.377,-56.772,-178.090,6.503,148.625
C08999=1185.063,172.627,-56.795,-178.087,6.504,148.625
C09000=1185.059,172.876,-56.817,-178.085,6.506,148.624
C09001=1185.054,173.125,-56.838,-178.082,6.508,148.624
C09002=1185.049,173.374,-56.862,-178.079,6.510,148.624
C09003=1185.044,173.622,-56.883,-178.077,6.511,148.623
C09004=1185.040,173.872,-56.905,-178.074,6.513,148.623
C09005=1185.035,174.121,-56.929,-178.071,6.515,148.623
C09006=1185.030,174.369,-56.950,-178.069,6.517,148.622
C09007=1185.026,174.618,-56.974,-178.066,6.519,148.622
C09008=1185.021,174.867,-56.995,-178.063,6.520,148.622
C09009=1185.016,175.116,-57.018,-178.061,6.522,148.621
C09010=1185.012,175.365,-57.041,-178.058,6.524,148.621
C09011=1185.007,175.614,-57.063,-178.055,6.526,148.620
C09012=1185.003,175.863,-57.085,-178.053,6.528,148.620
C09013=1184.998,176.112,-57.108,-178.050,6.529,148.620
C09014=1184.993,176.360,-57.130,-178.047,6.531,148.619
C09015=1184.988,176.610,-57.153,-178.045,6.533,148.619
C09016=1184.984,176.859,-57.175,-178.042,6.535,148.619
C09017=1184.979,177.108,-57.198,-178.040,6.537,148.619
C09018=1184.975,177.357,-57.220,-178.037,6.539,148.618
C09019=1184.971,177.606,-57.243,-178.034,6.540,148.618
C09020=1184.965,177.855,-57.265,-178.032,6.542,148.617
C09021=1184.961,178.103,-57.288,-178.029,6.544,148.617
C09022=1184.956,178.352,-57.311,-178.026,6.546,148.617
C09023=1184.951,178.601,-57.333,-178.024,6.547,148.616
C09024=1184.947,178.850,-57.356,-178.021,6.549,148.616
C09025=1184.942,179.099,-57.378,-178.018,6.551,148.616
C09026=1184.937,179.348,-57.401,-178.016,6.553,148.615
C09027=1184.933,179.597,-57.423,-178.013,6.555,148.615
C09028=1184.928,179.846,-57.447,-178.010,6.557,148.615
C09029=1184.924,180.095,-57.470,-178.007,6.559,148.614
C09030=1184.919,180.344,-57.492,-178.005,6.561,148.614
C09031=1184.915,180.592,-57.515,-178.002,6.563,148.613
C09032=1184.910,180.842,-57.538,-177.999,6.564,148.613
C09033=1184.905,181.091,-57.561,-177.996,6.566,148.613
C09034=1184.900,181.339,-57.583,-177.994,6.568,148.613
C09035=1184.896,181.588,-57.606,-177.992,6.570,148.612
C09036=1184.891,181.838,-57.628,-177.989,6.572,148.612
C09037=1184.887,182.087,-57.652,-177.986,6.574,148.612
C09038=1184.882,182.335,-57.674,-177.984,6.575,148.611
C09039=1184.877,182.584,-57.697,-177.981,6.577,148.611
C09040=1184.872,182.833,-57.720,-177.978,6.579,148.610
C09041=1184.869,183.082,-57.743,-177.976,6.581,148.610
C09042=1184.864,183.331,-57.766,-177.973,6.583,148.610
C09043=1184.859,183.579,-57.789,-177.970,6.584,148.609
C09044=1184.854,183.829,-57.811,-177.968,6.586,148.609
C09045=1184.850,184.078,-57.835,-177.965,6.588,148.609
C09046=1184.845,184.347,-57.859,-177.962,6.591,148.608
C09047=1184.840,184.617,-57.884,-177.959,6.592,148.608
C09048=1184.835,184.886,-57.910,-177.956,6.594,148.608
C09049=1184.830,185.156,-57.934,-177.953,6.597,148.607
C09050=1184.825,185.405,-57.958,-177.950,6.599,148.607
C09051=1184.820,185.654,-57.980,-177.948,6.601,148.607
C09052=1184.816,185.902,-58.003,-177.946,6.602,148.606
C09053=1184.811,186.151,-58.026,-177.943,6.604,148.606
C09054=1184.806,186.400,-58.049,-177.940,6.606,148.606
C09055=1184.802,186.649,-58.073,-177.938,6.608,148.605
C09056=1184.798,186.898,-58.096,-177.935,6.610,148.605
C09057=1184.793,187.147,-58.119,-177.932,6.612,148.605
C09058=1184.788,187.396,-58.142,-177.929,6.614,148.604
C09059=1184.783,187.644,-58.165,-177.926,6.616,148.604
C09060=1184.779,187.893,-58.188,-177.924,6.618,148.604
C09061=1184.774,188.142,-58.211,-177.921,6.620,148.604
C09062=1184.770,188.391,-58.235,-177.919,6.621,148.603
C09063=1184.765,188.640,-58.258,-177.916,6.623,148.603
C09064=1184.761,188.889,-58.281,-177.913,6.625,148.602
C09065=1184.756,189.138,-58.304,-177.911,6.627,148.602
C09066=1184.752,189.387,-58.328,-177.908,6.629,148.602
C09067=1184.746,189.635,-58.351,-177.905,6.631,148.601
C09068=1184.742,189.884,-58.374,-177.903,6.633,148.601
C09069=1184.737,190.133,-58.397,-177.900,6.635,148.601
C09070=1184.733,190.382,-58.420,-177.897,6.637,148.601
C09071=1184.728,190.631,-58.443,-177.895,6.639,148.600
C09072=1184.724,190.880,-58.467,-177.892,6.641,148.600
C09073=1184.719,191.129,-58.491,-177.889,6.642,148.600
C09074=1184.714,191.378,-58.514,-177.887,6.644,148.599
C09075=1184.710,191.627,-58.538,-177.884,6.646,148.599
C09076=1184.705,191.876,-58.561,-177.881,6.649,148.599
C09077=1184.700,192.125,-58.584,-177.879,6.651,148.598
C09078=1184.696,192.374,-58.608,-177.876,6.652,148.598
C09079=1184.692,192.622,-58.631,-177.873,6.654,148.598
C09080=1184.687,192.871,-58.654,-177.871,6.656,148.597
C09081=1184.683,193.120,-58.678,-177.868,6.658,148.597
C09082=1184.678,193.369,-58.701,-177.866,6.660,148.597
C09083=1184.673,193.618,-58.725,-177.863,6.663,148.597
C09084=1184.668,193.866,-58.748,-177.860,6.664,148.596
C09085=1184.663,194.115,-58.772,-177.857,6.666,148.596
C09086=1184.659,194.364,-58.795,-177.855,6.668,148.595
C09087=1184.654,194.613,-58.818,-177.852,6.670,148.595
C09088=1184.650,194.861,-58.842,-177.850,6.672,148.595
C09089=1184.645,195.110,-58.866,-177.847,6.674,148.595
C09090=1184.640,195.359,-58.889,-177.844,6.676,148.594
C09091=1184.637,195.608,-58.914,-177.841,6.678,148.594
C09092=1184.632,195.858,-58.937,-177.838,6.680,148.594
C09093=1184.627,196.107,-58.960,-177.836,6.682,148.594
C09094=1184.623,196.355,-58.984,-177.834,6.684,148.593
C09095=1184.618,196.604,-59.008,-177.831,6.686,148.593
C09096=1184.614,196.852,-59.032,-177.828,6.688,148.593
C09097=1184.609,197.101,-59.055,-177.825,6.690,148.592
C09098=1184.604,197.350,-59.079,-177.823,6.692,148.592
C09099=1184.600,197.599,-59.103,-177.820,6.694,148.592
C09100=1184.595,197.848,-59.126,-177.817,6.696,148.591
C09101=1184.591,198.096,-59.150,-177.815,6.698,148.591
C09102=1184.585,198.346,-59.174,-177.812,6.699,148.591
C09103=1184.581,198.594,-59.198,-177.809,6.702,148.591
C09104=1184.576,198.843,-59.221,-177.807,6.704,148.590
C09105=1184.572,199.092,-59.246,-177.804,6.706,148.590
C09106=1184.567,199.341,-59.269,-177.801,6.708,148.589
C09107=1184.563,199.589,-59.293,-177.799,6.710,148.589
C09108=1184.559,199.839,-59.317,-177.796,6.712,148.589
C09109=1184.554,200.087,-59.341,-177.793,6.714,148.589
C09110=1184.550,200.336,-59.364,-177.791,6.716,148.588
C09111=1184.544,200.585,-59.389,-177.788,6.718,148.588
C09112=1184.540,200.834,-59.412,-177.786,6.720,148.588
C09113=1184.535,201.082,-59.436,-177.783,6.722,148.588
C09114=1184.531,201.331,-59.460,-177.780,6.724,148.587
C09115=1184.526,201.580,-59.484,-177.777,6.726,148.587
C09116=1184.522,201.829,-59.508,-177.775,6.728,148.587
C09117=1184.517,202.078,-59.532,-177.772,6.730,148.586
C09118=1184.513,202.327,-59.556,-177.770,6.732,148.586
C09119=1184.508,202.575,-59.580,-177.767,6.735,148.586
C09120=1184.503,202.824,-59.604,-177.764,6.736,148.585
C09121=1184.498,203.073,-59.628,-177.762,6.739,148.585
C09122=1184.495,203.322,-59.653,-177.759,6.740,148.585
C09123=1184.490,203.571,-59.676,-177.756,6.742,148.585
C09124=1184.485,203.819,-59.700,-177.753,6.745,148.584
C09125=1184.480,204.068,-59.725,-177.751,6.747,148.584
C09126=1184.476,204.317,-59.748,-177.748,6.749,148.584
C09127=1184.471,204.566,-59.772,-177.746,6.750,148.583
C09128=1184.467,204.815,-59.797,-177.742,6.753,148.583
C09129=1184.462,205.063,-59.821,-177.740,6.755,148.583
C09130=1184.458,205.312,-59.845,-177.738,6.757,148.583
C09131=1184.453,205.561,-59.869,-177.735,6.759,148.582
C09132=1184.448,205.810,-59.893,-177.732,6.761,148.582
C09133=1184.444,206.059,-59.918,-177.729,6.764,148.582
C09134=1184.440,206.307,-59.942,-177.727,6.765,148.582
C09135=1184.435,206.556,-59.967,-177.724,6.767,148.581
C09136=1184.430,206.805,-59.990,-177.722,6.769,148.581
C09137=1184.426,207.054,-60.014,-177.719,6.772,148.581
C09138=1184.421,207.303,-60.039,-177.716,6.774,148.580
C09139=1184.417,207.551,-60.063,-177.713,6.776,148.580
C09140=1184.412,207.799,-60.087,-177.711,6.777,148.580
C09141=1184.408,208.049,-60.112,-177.708,6.780,148.580
